LIN {X 0,Y 671.666,Z 913.822,A -85,B 0,C 180,E1 31372.923,E2 31372.923} C_VEL
LIN {X 0,Y 672.94,Z 893.638,A -85,B 0,C 180,E1 31372.091,E2 31372.091} C_VEL
LIN {X 0,Y 674.079,Z 873.149,A -85,B 0,C 180,E1 31371.357,E2 31371.357} C_VEL
LIN {X 0,Y 675.288,Z 850.138,A -85,B 0,C 180,E1 31370.661,E2 31370.661} C_VEL
LIN {X 0,Y 676.492,Z 822.718,A -85,B 0,C 180,E1 31370.003,E2 31370.003} C_VEL
LIN {X 0,Y 677.288,Z 796.769,A -85,B 0,C 180,E1 31369.548,E2 31369.548} C_VEL
LIN {X 0,Y 680.414,Z 579.65,A -85,B 0,C 180,E1 31366.739,E2 31366.739} C_VEL
LIN {X 0,Y 683.518,Z 369.829,A -85,B 0,C 180,E1 31363.955,E2 31363.955} C_VEL
LIN {X 0,Y 683.506,Z 361.175,A -85,B 0,C 180,E1 31363.826,E2 31363.826} C_VEL
LIN {X 0,Y 671.201,Z 343.19,A -85,B 0,C 180,E1 31362.442,E2 31362.442} C_VEL
LIN {X 0,Y 666.717,Z 337.316,A -85,B 0,C 180,E1 31361.923,E2 31361.923} C_VEL
LIN {X 0,Y 663.783,Z 333.148,A -85,B 0,C 180,E1 31361.571,E2 31361.571} C_VEL
LIN {X 0,Y 661.006,Z 329.319,A -85,B 0,C 180,E1 31361.235,E2 31361.235} C_VEL
LIN {X 0,Y 660.134,Z 328.105,A -85,B 0,C 180,E1 31361.129,E2 31361.129} C_VEL
LIN {X 0,Y 657.606,Z 325.421,A -85,B 0,C 180,E1 31360.83,E2 31360.83} C_VEL
LIN {X 0,Y 656.61,Z 322.443,A -85,B 0,C 180,E1 31360.675,E2 31360.675} C_VEL
LIN {X 0,Y 656.617,Z 322.441,A -85,B 0,C 180,E1 31358.189,E2 31358.189} C_VEL
LIN {X 0,Y 656.632,Z 322.413,A -85,B 0,C 180,E1 31355.035,E2 31355.035} C_VEL
LIN {X 0,Y 656.601,Z 322.44,A -85,B 0,C 180,E1 31352.311,E2 31352.311} C_VEL
LIN {X 0,Y 656.685,Z 322.411,A -85,B 0,C 180,E1 31349.435,E2 31349.435} C_VEL
LIN {X 0,Y 656.609,Z 322.425,A -85,B 0,C 180,E1 31346.443,E2 31346.443} C_VEL
LIN {X 0,Y 656.627,Z 322.43,A -85,B 0,C 180,E1 31343.799,E2 31343.799} C_VEL
LIN {X 0,Y 656.633,Z 322.407,A -85,B 0,C 180,E1 31340.595,E2 31340.595} C_VEL
LIN {X 0,Y 656.618,Z 322.434,A -85,B 0,C 180,E1 31338.007,E2 31338.007} C_VEL
LIN {X 0,Y 656.701,Z 322.403,A -85,B 0,C 180,E1 31335.092,E2 31335.092} C_VEL
LIN {X 0,Y 656.627,Z 322.434,A -85,B 0,C 180,E1 31332.131,E2 31332.131} C_VEL
LIN {X 0,Y 656.642,Z 322.414,A -85,B 0,C 180,E1 31329.466,E2 31329.466} C_VEL
LIN {X 0,Y 656.646,Z 322.432,A -85,B 0,C 180,E1 31326.207,E2 31326.207} C_VEL
LIN {X 0,Y 656.634,Z 322.418,A -85,B 0,C 180,E1 31323.579,E2 31323.579} C_VEL
LIN {X 0,Y 656.71,Z 322.429,A -85,B 0,C 180,E1 31320.523,E2 31320.523} C_VEL
LIN {X 0,Y 656.638,Z 322.42,A -85,B 0,C 180,E1 31317.644,E2 31317.644} C_VEL
LIN {X 0,Y 656.706,Z 322.421,A -85,B 0,C 180,E1 31314.706,E2 31314.706} C_VEL
LIN {X 0,Y 656.648,Z 322.417,A -85,B 0,C 180,E1 31311.682,E2 31311.682} C_VEL
LIN {X 0,Y 656.68,Z 322.422,A -85,B 0,C 180,E1 31308.85,E2 31308.85} C_VEL
LIN {X 0,Y 656.663,Z 322.41,A -85,B 0,C 180,E1 31305.719,E2 31305.719} C_VEL
LIN {X 0,Y 656.668,Z 322.428,A -85,B 0,C 180,E1 31302.91,E2 31302.91} C_VEL
LIN {X 0,Y 656.678,Z 322.403,A -85,B 0,C 180,E1 31299.686,E2 31299.686} C_VEL
LIN {X 0,Y 656.674,Z 322.435,A -85,B 0,C 180,E1 31296.773,E2 31296.773} C_VEL
LIN {X 0,Y 656.686,Z 322.424,A -85,B 0,C 180,E1 31293.544,E2 31293.544} C_VEL
LIN {X 0,Y 656.685,Z 322.409,A -85,B 0,C 180,E1 31290.54,E2 31290.54} C_VEL
LIN {X 0,Y 656.686,Z 322.425,A -85,B 0,C 180,E1 31287.35,E2 31287.35} C_VEL
LIN {X 0,Y 656.698,Z 322.433,A -85,B 0,C 180,E1 31284.327,E2 31284.327} C_VEL
LIN {X 0,Y 656.736,Z 322.619,A -85,B 0,C 180,E1 31281.555,E2 31281.555} C_VEL
LIN {X 0,Y 658.039,Z 325.986,A -85,B 0,C 180,E1 31281.13,E2 31281.13} C_VEL
LIN {X 0,Y 659.196,Z 328.329,A -85,B 0,C 180,E1 31280.812,E2 31280.812} C_VEL
LIN {X 0,Y 663.314,Z 336.664,A -85,B 0,C 180,E1 31279.705,E2 31279.705} C_VEL
LIN {X 0,Y 670.239,Z 350.9,A -85,B 0,C 180,E1 31277.945,E2 31277.945} C_VEL
LIN {X 0,Y 680.871,Z 366.63,A -85,B 0,C 180,E1 31276.729,E2 31276.729} C_VEL
LIN {X 0,Y 683.852,Z 379.489,A -85,B 0,C 180,E1 31276.273,E2 31276.273} C_VEL
LIN {X 0,Y 680.729,Z 587.028,A -85,B 0,C 180,E1 31273.513,E2 31273.513} C_VEL
LIN {X 0,Y 677.649,Z 809.677,A -85,B 0,C 180,E1 31270.64,E2 31270.64} C_VEL
LIN {X 0,Y 676.889,Z 840.625,A -85,B 0,C 180,E1 31270.183,E2 31270.183} C_VEL
LIN {X 0,Y 675.965,Z 864.916,A -85,B 0,C 180,E1 31269.679,E2 31269.679} C_VEL
LIN {X 0,Y 674.842,Z 889.591,A -85,B 0,C 180,E1 31269.027,E2 31269.027} C_VEL
LIN {X 0,Y 673.329,Z 917.024,A -85,B 0,C 180,E1 31268.116,E2 31268.116} C_VEL
LIN {X 0,Y 671.946,Z 939.064,A -85,B 0,C 180,E1 31267.24,E2 31267.24} C_VEL
LIN {X 0,Y 670.562,Z 959.722,A -85,B 0,C 180,E1 31266.296,E2 31266.296} C_VEL
LIN {X 0,Y 669.028,Z 981.503,A -85,B 0,C 180,E1 31265.163,E2 31265.163} C_VEL
LIN {X 0,Y 667.169,Z 1006.405,A -85,B 0,C 180,E1 31263.676,E2 31263.676} C_VEL
LIN {X 0,Y 665.527,Z 1027.238,A -85,B 0,C 180,E1 31262.257,E2 31262.257} C_VEL
LIN {X 0,Y 664.066,Z 1046.482,A -85,B 0,C 180,E1 31260.792,E2 31260.792} C_VEL
LIN {X 0,Y 662.377,Z 1069.251,A -85,B 0,C 180,E1 31258.835,E2 31258.835} C_VEL
LIN {X 0,Y 661.095,Z 1086.391,A -85,B 0,C 180,E1 31257.178,E2 31257.178} C_VEL
LIN {X 0,Y 659.976,Z 1103.08,A -85,B 0,C 180,E1 31255.388,E2 31255.388} C_VEL
LIN {X 0,Y 658.84,Z 1120.853,A -85,B 0,C 180,E1 31253.24,E2 31253.24} C_VEL
LIN {X 0,Y 658.05,Z 1134.796,A -85,B 0,C 180,E1 31251.339,E2 31251.339} C_VEL
LIN {X 0,Y 657.408,Z 1147.739,A -85,B 0,C 180,E1 31249.363,E2 31249.363} C_VEL
LIN {X 0,Y 656.816,Z 1161.282,A -85,B 0,C 180,E1 31246.994,E2 31246.994} C_VEL
LIN {X 0,Y 656.46,Z 1171.486,A -85,B 0,C 180,E1 31244.916,E2 31244.916} C_VEL
LIN {X 0,Y 656.243,Z 1179.514,A -85,B 0,C 180,E1 31243.032,E2 31243.032} C_VEL
LIN {X 0,Y 656.056,Z 1187.306,A -85,B 0,C 180,E1 31240.893,E2 31240.893} C_VEL
LIN {X 0,Y 655.979,Z 1194.036,A -85,B 0,C 180,E1 31238.591,E2 31238.591} C_VEL
LIN {X 0,Y 655.933,Z 1199.09,A -85,B 0,C 180,E1 31236.301,E2 31236.301} C_VEL
LIN {X 0,Y 655.917,Z 1202.479,A -85,B 0,C 180,E1 31234.108,E2 31234.108} C_VEL
LIN {X 0,Y 655.907,Z 1204.549,A -85,B 0,C 180,E1 31231.747,E2 31231.747} C_VEL
LIN {X 0,Y 655.891,Z 1204.872,A -85,B 0,C 180,E1 31229.476,E2 31229.476} C_VEL
LIN {X 0,Y 655.908,Z 1203.947,A -85,B 0,C 180,E1 31227.379,E2 31227.379} C_VEL
LIN {X 0,Y 655.919,Z 1201.428,A -85,B 0,C 180,E1 31225.103,E2 31225.103} C_VEL
LIN {X 0,Y 655.949,Z 1197.152,A -85,B 0,C 180,E1 31222.732,E2 31222.732} C_VEL
LIN {X 0,Y 656.009,Z 1191.376,A -85,B 0,C 180,E1 31220.437,E2 31220.437} C_VEL
LIN {X 0,Y 656.126,Z 1184.279,A -85,B 0,C 180,E1 31218.217,E2 31218.217} C_VEL
LIN {X 0,Y 656.39,Z 1174.089,A -85,B 0,C 180,E1 31215.658,E2 31215.658} C_VEL
LIN {X 0,Y 656.694,Z 1164.273,A -85,B 0,C 180,E1 31213.587,E2 31213.587} C_VEL
LIN {X 0,Y 657.112,Z 1154.137,A -85,B 0,C 180,E1 31211.716,E2 31211.716} C_VEL
LIN {X 0,Y 657.764,Z 1140.78,A -85,B 0,C 180,E1 31209.536,E2 31209.536} C_VEL
LIN {X 0,Y 658.6,Z 1125.104,A -85,B 0,C 180,E1 31207.318,E2 31207.318} C_VEL
LIN {X 0,Y 659.476,Z 1110.399,A -85,B 0,C 180,E1 31205.467,E2 31205.467} C_VEL
LIN {X 0,Y 660.73,Z 1092.314,A -85,B 0,C 180,E1 31203.428,E2 31203.428} C_VEL
LIN {X 0,Y 662,Z 1073.819,A -85,B 0,C 180,E1 31201.591,E2 31201.591} C_VEL
LIN {X 0,Y 663.289,Z 1056.842,A -85,B 0,C 180,E1 31200.069,E2 31200.069} C_VEL
LIN {X 0,Y 664.963,Z 1035.53,A -85,B 0,C 180,E1 31198.348,E2 31198.348} C_VEL
LIN {X 0,Y 666.618,Z 1013.004,A -85,B 0,C 180,E1 31196.756,E2 31196.756} C_VEL
LIN {X 0,Y 668.131,Z 993.022,A -85,B 0,C 180,E1 31195.499,E2 31195.499} C_VEL
LIN {X 0,Y 669.972,Z 968.967,A -85,B 0,C 180,E1 31194.161,E2 31194.161} C_VEL
LIN {X 0,Y 671.656,Z 944.002,A -85,B 0,C 180,E1 31192.976,E2 31192.976} C_VEL
LIN {X 0,Y 672.974,Z 923.056,A -85,B 0,C 180,E1 31192.114,E2 31192.114} C_VEL
LIN {X 0,Y 674.098,Z 902.837,A -85,B 0,C 180,E1 31191.392,E2 31191.392} C_VEL
LIN {X 0,Y 675.317,Z 879.538,A -85,B 0,C 180,E1 31190.689,E2 31190.689} C_VEL
LIN {X 0,Y 676.525,Z 851.65,A -85,B 0,C 180,E1 31190.026,E2 31190.026} C_VEL
LIN {X 0,Y 677.299,Z 826.243,A -85,B 0,C 180,E1 31189.585,E2 31189.585} C_VEL
LIN {X 0,Y 680.398,Z 610.207,A -85,B 0,C 180,E1 31186.79,E2 31186.79} C_VEL
LIN {X 0,Y 683.523,Z 400.862,A -85,B 0,C 180,E1 31184.016,E2 31184.016} C_VEL
LIN {X 0,Y 683.703,Z 378.044,A -85,B 0,C 180,E1 31183.693,E2 31183.693} C_VEL
LIN {X 0,Y 680.509,Z 365.883,A -85,B 0,C 180,E1 31183.227,E2 31183.227} C_VEL
LIN {X 0,Y 669.705,Z 349.983,A -85,B 0,C 180,E1 31181.969,E2 31181.969} C_VEL
LIN {X 0,Y 661.964,Z 333.955,A -85,B 0,C 180,E1 31179.938,E2 31179.938} C_VEL
LIN {X 0,Y 659.979,Z 329.954,A -85,B 0,C 180,E1 31179.405,E2 31179.405} C_VEL
LIN {X 0,Y 658.426,Z 326.508,A -85,B 0,C 180,E1 31178.955,E2 31178.955} C_VEL
LIN {X 0,Y 656.846,Z 323.199,A -85,B 0,C 180,E1 31178.507,E2 31178.507} C_VEL
LIN {X 0,Y 656.707,Z 322.413,A -85,B 0,C 180,E1 31178.405,E2 31178.405} C_VEL
LIN {X 0,Y 656.675,Z 322.429,A -85,B 0,C 180,E1 31175.302,E2 31175.302} C_VEL
LIN {X 0,Y 656.707,Z 322.423,A -85,B 0,C 180,E1 31172.305,E2 31172.305} C_VEL
LIN {X 0,Y 656.672,Z 322.412,A -85,B 0,C 180,E1 31169.255,E2 31169.255} C_VEL
LIN {X 0,Y 656.703,Z 322.418,A -85,B 0,C 180,E1 31166.263,E2 31166.263} C_VEL
LIN {X 0,Y 656.672,Z 322.434,A -85,B 0,C 180,E1 31163.124,E2 31163.124} C_VEL
LIN {X 0,Y 656.698,Z 322.401,A -85,B 0,C 180,E1 31160.127,E2 31160.127} C_VEL
LIN {X 0,Y 656.666,Z 322.429,A -85,B 0,C 180,E1 31156.999,E2 31156.999} C_VEL
LIN {X 0,Y 656.682,Z 322.407,A -85,B 0,C 180,E1 31154.096,E2 31154.096} C_VEL
LIN {X 0,Y 656.668,Z 322.424,A -85,B 0,C 180,E1 31150.972,E2 31150.972} C_VEL
LIN {X 0,Y 656.659,Z 322.414,A -85,B 0,C 180,E1 31148.141,E2 31148.141} C_VEL
LIN {X 0,Y 656.677,Z 322.422,A -85,B 0,C 180,E1 31144.979,E2 31144.979} C_VEL
LIN {X 0,Y 656.646,Z 322.416,A -85,B 0,C 180,E1 31142.182,E2 31142.182} C_VEL
LIN {X 0,Y 656.705,Z 322.424,A -85,B 0,C 180,E1 31139.128,E2 31139.128} C_VEL
LIN {X 0,Y 656.635,Z 322.417,A -85,B 0,C 180,E1 31136.246,E2 31136.246} C_VEL
LIN {X 0,Y 656.699,Z 322.43,A -85,B 0,C 180,E1 31133.355,E2 31133.355} C_VEL
LIN {X 0,Y 656.637,Z 322.414,A -85,B 0,C 180,E1 31130.357,E2 31130.357} C_VEL
LIN {X 0,Y 656.64,Z 322.433,A -85,B 0,C 180,E1 31127.691,E2 31127.691} C_VEL
LIN {X 0,Y 656.66,Z 322.411,A -85,B 0,C 180,E1 31124.543,E2 31124.543} C_VEL
LIN {X 0,Y 656.624,Z 322.434,A -85,B 0,C 180,E1 31121.81,E2 31121.81} C_VEL
LIN {X 0,Y 656.707,Z 322.404,A -85,B 0,C 180,E1 31118.847,E2 31118.847} C_VEL
LIN {X 0,Y 656.619,Z 322.43,A -85,B 0,C 180,E1 31115.914,E2 31115.914} C_VEL
LIN {X 0,Y 656.63,Z 322.422,A -85,B 0,C 180,E1 31113.307,E2 31113.307} C_VEL
LIN {X 0,Y 656.637,Z 322.411,A -85,B 0,C 180,E1 31110.136,E2 31110.136} C_VEL
LIN {X 0,Y 656.609,Z 322.439,A -85,B 0,C 180,E1 31107.523,E2 31107.523} C_VEL
LIN {X 0,Y 656.676,Z 322.411,A -85,B 0,C 180,E1 31104.647,E2 31104.647} C_VEL
LIN {X 0,Y 656.604,Z 322.415,A -85,B 0,C 180,E1 31101.649,E2 31101.649} C_VEL
LIN {X 0,Y 656.688,Z 322.418,A -85,B 0,C 180,E1 31100.473,E2 31100.473} C_VEL
LIN {X 0,Y 656.825,Z 323.195,A -85,B 0,C 180,E1 31100.104,E2 31100.104} C_VEL
LIN {X 0,Y 657.18,Z 325.756,A -85,B 0,C 180,E1 31099.685,E2 31099.685} C_VEL
LIN {X 0,Y 658.094,Z 331.001,A -85,B 0,C 180,E1 31099.187,E2 31099.187} C_VEL
LIN {X 0,Y 660.809,Z 339.923,A -85,B 0,C 180,E1 31098.553,E2 31098.553} C_VEL
LIN {X 0,Y 663.684,Z 344.552,A -85,B 0,C 180,E1 31098.166,E2 31098.166} C_VEL
LIN {X 0,Y 670.686,Z 354.26,A -85,B 0,C 180,E1 31097.344,E2 31097.344} C_VEL
LIN {X 0,Y 678.016,Z 365.563,A -85,B 0,C 180,E1 31096.503,E2 31096.503} C_VEL
LIN {X 0,Y 674.796,Z 565.744,A -85,B 0,C 180,E1 31093.822,E2 31093.822} C_VEL
LIN {X 0,Y 671.317,Z 791.977,A -85,B 0,C 180,E1 31090.876,E2 31090.876} C_VEL
LIN {X 0,Y 670.56,Z 815.572,A -85,B 0,C 180,E1 31090.489,E2 31090.489} C_VEL
LIN {X 0,Y 669.499,Z 841.04,A -85,B 0,C 180,E1 31089.93,E2 31089.93} C_VEL
LIN {X 0,Y 668.036,Z 868.498,A -85,B 0,C 180,E1 31089.141,E2 31089.141} C_VEL
LIN {X 0,Y 666.707,Z 890.267,A -85,B 0,C 180,E1 31088.38,E2 31088.38} C_VEL
LIN {X 0,Y 665.306,Z 910.812,A -85,B 0,C 180,E1 31087.547,E2 31087.547} C_VEL
LIN {X 0,Y 663.778,Z 931.891,A -85,B 0,C 180,E1 31086.566,E2 31086.566} C_VEL
LIN {X 0,Y 661.891,Z 956.652,A -85,B 0,C 180,E1 31085.243,E2 31085.243} C_VEL
LIN {X 0,Y 659.976,Z 979.437,A -85,B 0,C 180,E1 31083.832,E2 31083.832} C_VEL
LIN {X 0,Y 658.322,Z 998.997,A -85,B 0,C 180,E1 31082.472,E2 31082.472} C_VEL
LIN {X 0,Y 656.56,Z 1020.781,A -85,B 0,C 180,E1 31080.776,E2 31080.776} C_VEL
LIN {X 0,Y 654.855,Z 1041.333,A -85,B 0,C 180,E1 31078.947,E2 31078.947} C_VEL
LIN {X 0,Y 653.526,Z 1057.819,A -85,B 0,C 180,E1 31077.321,E2 31077.321} C_VEL
LIN {X 0,Y 652.214,Z 1076.039,A -85,B 0,C 180,E1 31075.322,E2 31075.322} C_VEL
LIN {X 0,Y 651.029,Z 1092.653,A -85,B 0,C 180,E1 31073.247,E2 31073.247} C_VEL
LIN {X 0,Y 650.204,Z 1106.086,A -85,B 0,C 180,E1 31071.374,E2 31071.374} C_VEL
LIN {X 0,Y 649.455,Z 1120.323,A -85,B 0,C 180,E1 31069.143,E2 31069.143} C_VEL
LIN {X 0,Y 648.84,Z 1132.921,A -85,B 0,C 180,E1 31066.84,E2 31066.84} C_VEL
LIN {X 0,Y 648.504,Z 1142.107,A -85,B 0,C 180,E1 31064.92,E2 31064.92} C_VEL
LIN {X 0,Y 648.255,Z 1150.555,A -85,B 0,C 180,E1 31062.884,E2 31062.884} C_VEL
LIN {X 0,Y 648.065,Z 1158.619,A -85,B 0,C 180,E1 31060.579,E2 31060.579} C_VEL
LIN {X 0,Y 647.974,Z 1165.226,A -85,B 0,C 180,E1 31058.161,E2 31058.161} C_VEL
LIN {X 0,Y 647.931,Z 1169.805,A -85,B 0,C 180,E1 31055.934,E2 31055.934} C_VEL
LIN {X 0,Y 647.913,Z 1173.144,A -85,B 0,C 180,E1 31053.539,E2 31053.539} C_VEL
LIN {X 0,Y 647.91,Z 1174.68,A -85,B 0,C 180,E1 31051.238,E2 31051.238} C_VEL
LIN {X 0,Y 647.896,Z 1174.838,A -85,B 0,C 180,E1 31049.293,E2 31049.293} C_VEL
LIN {X 0,Y 647.909,Z 1173.911,A -85,B 0,C 180,E1 31047.258,E2 31047.258} C_VEL
LIN {X 0,Y 647.921,Z 1171.367,A -85,B 0,C 180,E1 31044.954,E2 31044.954} C_VEL
LIN {X 0,Y 647.946,Z 1167.055,A -85,B 0,C 180,E1 31042.552,E2 31042.552} C_VEL
LIN {X 0,Y 648.019,Z 1161.246,A -85,B 0,C 180,E1 31040.228,E2 31040.228} C_VEL
LIN {X 0,Y 648.159,Z 1153.801,A -85,B 0,C 180,E1 31037.89,E2 31037.89} C_VEL
LIN {X 0,Y 648.461,Z 1143.728,A -85,B 0,C 180,E1 31035.353,E2 31035.353} C_VEL
LIN {X 0,Y 648.781,Z 1134.303,A -85,B 0,C 180,E1 31033.343,E2 31033.343} C_VEL
LIN {X 0,Y 649.238,Z 1123.964,A -85,B 0,C 180,E1 31031.41,E2 31031.41} C_VEL
LIN {X 0,Y 649.968,Z 1110.475,A -85,B 0,C 180,E1 31029.185,E2 31029.185} C_VEL
LIN {X 0,Y 650.893,Z 1094.731,A -85,B 0,C 180,E1 31026.939,E2 31026.939} C_VEL
LIN {X 0,Y 651.841,Z 1080.663,A -85,B 0,C 180,E1 31025.147,E2 31025.147} C_VEL
LIN {X 0,Y 653.205,Z 1062.368,A -85,B 0,C 180,E1 31023.058,E2 31023.058} C_VEL
LIN {X 0,Y 654.644,Z 1043.712,A -85,B 0,C 180,E1 31021.187,E2 31021.187} C_VEL
LIN {X 0,Y 656.036,Z 1026.779,A -85,B 0,C 180,E1 31019.653,E2 31019.653} C_VEL
LIN {X 0,Y 657.802,Z 1006.081,A -85,B 0,C 180,E1 31017.962,E2 31017.962} C_VEL
LIN {X 0,Y 659.644,Z 983.162,A -85,B 0,C 180,E1 31016.323,E2 31016.323} C_VEL
LIN {X 0,Y 661.323,Z 962.904,A -85,B 0,C 180,E1 31015.04,E2 31015.04} C_VEL
LIN {X 0,Y 663.335,Z 938.507,A -85,B 0,C 180,E1 31013.674,E2 31013.674} C_VEL
LIN {X 0,Y 665.121,Z 913.811,A -85,B 0,C 180,E1 31012.496,E2 31012.496} C_VEL
LIN {X 0,Y 666.501,Z 893.662,A -85,B 0,C 180,E1 31011.661,E2 31011.661} C_VEL
LIN {X 0,Y 667.739,Z 873.127,A -85,B 0,C 180,E1 31010.921,E2 31010.921} C_VEL
LIN {X 0,Y 669.012,Z 850.563,A -85,B 0,C 180,E1 31010.234,E2 31010.234} C_VEL
LIN {X 0,Y 670.3,Z 823.602,A -85,B 0,C 180,E1 31009.579,E2 31009.579} C_VEL
LIN {X 0,Y 671.173,Z 797.336,A -85,B 0,C 180,E1 31009.112,E2 31009.112} C_VEL
LIN {X 0,Y 674.494,Z 585.107,A -85,B 0,C 180,E1 31006.343,E2 31006.343} C_VEL
LIN {X 0,Y 677.899,Z 373.5,A -85,B 0,C 180,E1 31003.516,E2 31003.516} C_VEL
LIN {X 0,Y 677.911,Z 365.067,A -85,B 0,C 180,E1 31003.39,E2 31003.39} C_VEL
LIN {X 0,Y 667.133,Z 349.224,A -85,B 0,C 180,E1 31002.151,E2 31002.151} C_VEL
LIN {X 0,Y 659.308,Z 338.748,A -85,B 0,C 180,E1 31001.219,E2 31001.219} C_VEL
LIN {X 0,Y 656.27,Z 334.548,A -85,B 0,C 180,E1 31000.844,E2 31000.844} C_VEL
LIN {X 0,Y 653.322,Z 330.877,A -85,B 0,C 180,E1 31000.481,E2 31000.481} C_VEL
LIN {X 0,Y 652.237,Z 329.139,A -85,B 0,C 180,E1 31000.34,E2 31000.34} C_VEL
LIN {X 0,Y 649.752,Z 326.511,A -85,B 0,C 180,E1 31000.035,E2 31000.035} C_VEL
LIN {X 0,Y 648.72,Z 323.425,A -85,B 0,C 180,E1 30999.865,E2 30999.865} C_VEL
LIN {X 0,Y 648.678,Z 323.43,A -85,B 0,C 180,E1 30996.843,E2 30996.843} C_VEL
LIN {X 0,Y 648.663,Z 323.402,A -85,B 0,C 180,E1 30994.238,E2 30994.238} C_VEL
LIN {X 0,Y 648.729,Z 323.402,A -85,B 0,C 180,E1 30991.197,E2 30991.197} C_VEL
LIN {X 0,Y 648.669,Z 323.426,A -85,B 0,C 180,E1 30988.445,E2 30988.445} C_VEL
LIN {X 0,Y 648.686,Z 323.402,A -85,B 0,C 180,E1 30985.822,E2 30985.822} C_VEL
LIN {X 0,Y 648.69,Z 323.423,A -85,B 0,C 180,E1 30982.57,E2 30982.57} C_VEL
LIN {X 0,Y 648.675,Z 323.396,A -85,B 0,C 180,E1 30980.011,E2 30980.011} C_VEL
LIN {X 0,Y 648.766,Z 323.415,A -85,B 0,C 180,E1 30977.028,E2 30977.028} C_VEL
LIN {X 0,Y 648.682,Z 323.403,A -85,B 0,C 180,E1 30974.096,E2 30974.096} C_VEL
LIN {X 0,Y 648.717,Z 323.425,A -85,B 0,C 180,E1 30971.379,E2 30971.379} C_VEL
LIN {X 0,Y 648.702,Z 323.4,A -85,B 0,C 180,E1 30968.242,E2 30968.242} C_VEL
LIN {X 0,Y 648.697,Z 323.424,A -85,B 0,C 180,E1 30965.573,E2 30965.573} C_VEL
LIN {X 0,Y 648.748,Z 323.39,A -85,B 0,C 180,E1 30962.473,E2 30962.473} C_VEL
LIN {X 0,Y 648.698,Z 323.422,A -85,B 0,C 180,E1 30959.647,E2 30959.647} C_VEL
LIN {X 0,Y 648.763,Z 323.388,A -85,B 0,C 180,E1 30956.731,E2 30956.731} C_VEL
LIN {X 0,Y 648.708,Z 323.42,A -85,B 0,C 180,E1 30953.717,E2 30953.717} C_VEL
LIN {X 0,Y 648.74,Z 323.392,A -85,B 0,C 180,E1 30950.865,E2 30950.865} C_VEL
LIN {X 0,Y 648.722,Z 323.418,A -85,B 0,C 180,E1 30947.719,E2 30947.719} C_VEL
LIN {X 0,Y 648.728,Z 323.393,A -85,B 0,C 180,E1 30944.901,E2 30944.901} C_VEL
LIN {X 0,Y 648.734,Z 323.415,A -85,B 0,C 180,E1 30941.674,E2 30941.674} C_VEL
LIN {X 0,Y 648.736,Z 323.399,A -85,B 0,C 180,E1 30938.764,E2 30938.764} C_VEL
LIN {X 0,Y 648.744,Z 323.402,A -85,B 0,C 180,E1 30935.603,E2 30935.603} C_VEL
LIN {X 0,Y 648.751,Z 323.421,A -85,B 0,C 180,E1 30932.559,E2 30932.559} C_VEL
LIN {X 0,Y 648.738,Z 323.405,A -85,B 0,C 180,E1 30929.317,E2 30929.317} C_VEL
LIN {X 0,Y 648.759,Z 323.394,A -85,B 0,C 180,E1 30926.3,E2 30926.3} C_VEL
LIN {X 0,Y 648.739,Z 323.4,A -85,B 0,C 180,E1 30923.12,E2 30923.12} C_VEL
LIN {X 0,Y 648.774,Z 323.536,A -85,B 0,C 180,E1 30922.332,E2 30922.332} C_VEL
LIN {X 0,Y 649.998,Z 326.772,A -85,B 0,C 180,E1 30921.913,E2 30921.913} C_VEL
LIN {X 0,Y 651.055,Z 328.483,A -85,B 0,C 180,E1 30921.65,E2 30921.65} C_VEL
LIN {X 0,Y 659.144,Z 345.329,A -85,B 0,C 180,E1 30919.4,E2 30919.4} C_VEL
LIN {X 0,Y 661.685,Z 350.479,A -85,B 0,C 180,E1 30918.773,E2 30918.773} C_VEL
LIN {X 0,Y 675.933,Z 371.231,A -85,B 0,C 180,E1 30917.105,E2 30917.105} C_VEL
LIN {X 0,Y 678.28,Z 381.651,A -85,B 0,C 180,E1 30916.734,E2 30916.734} C_VEL
LIN {X 0,Y 674.888,Z 589.308,A -85,B 0,C 180,E1 30913.953,E2 30913.953} C_VEL
LIN {X 0,Y 671.538,Z 812.221,A -85,B 0,C 180,E1 30911.054,E2 30911.054} C_VEL
LIN {X 0,Y 670.725,Z 841.411,A -85,B 0,C 180,E1 30910.611,E2 30910.611} C_VEL
LIN {X 0,Y 669.756,Z 865.157,A -85,B 0,C 180,E1 30910.114,E2 30910.114} C_VEL
LIN {X 0,Y 668.563,Z 889.44,A -85,B 0,C 180,E1 30909.469,E2 30909.469} C_VEL
LIN {X 0,Y 666.876,Z 917.596,A -85,B 0,C 180,E1 30908.527,E2 30908.527} C_VEL
LIN {X 0,Y 665.363,Z 939.922,A -85,B 0,C 180,E1 30907.63,E2 30907.63} C_VEL
LIN {X 0,Y 663.854,Z 960.724,A -85,B 0,C 180,E1 30906.668,E2 30906.668} C_VEL
LIN {X 0,Y 662.096,Z 983.91,A -85,B 0,C 180,E1 30905.443,E2 30905.443} C_VEL
LIN {X 0,Y 660.055,Z 1008.607,A -85,B 0,C 180,E1 30903.932,E2 30903.932} C_VEL
LIN {X 0,Y 658.45,Z 1027.583,A -85,B 0,C 180,E1 30902.62,E2 30902.62} C_VEL
LIN {X 0,Y 656.822,Z 1047.088,A -85,B 0,C 180,E1 30901.118,E2 30901.118} C_VEL
LIN {X 0,Y 654.983,Z 1069.759,A -85,B 0,C 180,E1 30899.141,E2 30899.141} C_VEL
LIN {X 0,Y 653.646,Z 1086.39,A -85,B 0,C 180,E1 30897.513,E2 30897.513} C_VEL
LIN {X 0,Y 652.369,Z 1103.306,A -85,B 0,C 180,E1 30895.679,E2 30895.679} C_VEL
LIN {X 0,Y 651.106,Z 1121.566,A -85,B 0,C 180,E1 30893.436,E2 30893.436} C_VEL
LIN {X 0,Y 650.245,Z 1135.429,A -85,B 0,C 180,E1 30891.515,E2 30891.515} C_VEL
LIN {X 0,Y 649.487,Z 1149.548,A -85,B 0,C 180,E1 30889.313,E2 30889.313} C_VEL
LIN {X 0,Y 648.875,Z 1162.214,A -85,B 0,C 180,E1 30887.024,E2 30887.024} C_VEL
LIN {X 0,Y 648.512,Z 1171.487,A -85,B 0,C 180,E1 30885.103,E2 30885.103} C_VEL
LIN {X 0,Y 648.28,Z 1179.515,A -85,B 0,C 180,E1 30883.195,E2 30883.195} C_VEL
LIN {X 0,Y 648.084,Z 1187.034,A -85,B 0,C 180,E1 30881.112,E2 30881.112} C_VEL
LIN {X 0,Y 647.987,Z 1193.816,A -85,B 0,C 180,E1 30878.787,E2 30878.787} C_VEL
LIN {X 0,Y 647.935,Z 1199.101,A -85,B 0,C 180,E1 30876.372,E2 30876.372} C_VEL
LIN {X 0,Y 647.918,Z 1202.476,A -85,B 0,C 180,E1 30874.159,E2 30874.159} C_VEL
LIN {X 0,Y 647.907,Z 1204.549,A -85,B 0,C 180,E1 30871.769,E2 30871.769} C_VEL
LIN {X 0,Y 647.892,Z 1204.872,A -85,B 0,C 180,E1 30869.469,E2 30869.469} C_VEL
LIN {X 0,Y 647.909,Z 1203.944,A -85,B 0,C 180,E1 30867.346,E2 30867.346} C_VEL
LIN {X 0,Y 647.922,Z 1201.427,A -85,B 0,C 180,E1 30865.042,E2 30865.042} C_VEL
LIN {X 0,Y 647.951,Z 1197.151,A -85,B 0,C 180,E1 30862.641,E2 30862.641} C_VEL
LIN {X 0,Y 648.018,Z 1191.373,A -85,B 0,C 180,E1 30860.318,E2 30860.318} C_VEL
LIN {X 0,Y 648.146,Z 1184.279,A -85,B 0,C 180,E1 30858.07,E2 30858.07} C_VEL
LIN {X 0,Y 648.439,Z 1174.338,A -85,B 0,C 180,E1 30855.535,E2 30855.535} C_VEL
LIN {X 0,Y 648.771,Z 1164.544,A -85,B 0,C 180,E1 30853.434,E2 30853.434} C_VEL
LIN {X 0,Y 649.238,Z 1154.237,A -85,B 0,C 180,E1 30851.503,E2 30851.503} C_VEL
LIN {X 0,Y 649.924,Z 1141.364,A -85,B 0,C 180,E1 30849.372,E2 30849.372} C_VEL
LIN {X 0,Y 650.838,Z 1125.803,A -85,B 0,C 180,E1 30847.128,E2 30847.128} C_VEL
LIN {X 0,Y 651.804,Z 1111.152,A -85,B 0,C 180,E1 30845.252,E2 30845.252} C_VEL
LIN {X 0,Y 653.113,Z 1093.727,A -85,B 0,C 180,E1 30843.251,E2 30843.251} C_VEL
LIN {X 0,Y 654.547,Z 1074.832,A -85,B 0,C 180,E1 30841.337,E2 30841.337} C_VEL
LIN {X 0,Y 655.937,Z 1057.951,A -85,B 0,C 180,E1 30839.8,E2 30839.8} C_VEL
LIN {X 0,Y 657.511,Z 1039.194,A -85,B 0,C 180,E1 30838.254,E2 30838.254} C_VEL
LIN {X 0,Y 659.486,Z 1015.133,A -85,B 0,C 180,E1 30836.501,E2 30836.501} C_VEL
LIN {X 0,Y 661.141,Z 994.951,A -85,B 0,C 180,E1 30835.207,E2 30835.207} C_VEL
LIN {X 0,Y 662.831,Z 974.061,A -85,B 0,C 180,E1 30834.017,E2 30834.017} C_VEL
LIN {X 0,Y 664.822,Z 948.476,A -85,B 0,C 180,E1 30832.747,E2 30832.747} C_VEL
LIN {X 0,Y 666.407,Z 925.175,A -85,B 0,C 180,E1 30831.764,E2 30831.764} C_VEL
LIN {X 0,Y 667.661,Z 904.466,A -85,B 0,C 180,E1 30831.01,E2 30831.01} C_VEL
LIN {X 0,Y 668.911,Z 882.309,A -85,B 0,C 180,E1 30830.328,E2 30830.328} C_VEL
LIN {X 0,Y 670.161,Z 856.684,A -85,B 0,C 180,E1 30829.689,E2 30829.689} C_VEL
LIN {X 0,Y 671.133,Z 829.116,A -85,B 0,C 180,E1 30829.183,E2 30829.183} C_VEL
LIN {X 0,Y 672.991,Z 713.103,A -85,B 0,C 180,E1 30827.667,E2 30827.667} C_VEL
LIN {X 0,Y 676.466,Z 491.125,A -85,B 0,C 180,E1 30824.743,E2 30824.743} C_VEL
LIN {X 0,Y 678.142,Z 380.284,A -85,B 0,C 180,E1 30823.233,E2 30823.233} C_VEL
LIN {X 0,Y 675.637,Z 370.746,A -85,B 0,C 180,E1 30822.86,E2 30822.86} C_VEL
LIN {X 0,Y 661.182,Z 349.497,A -85,B 0,C 180,E1 30821.136,E2 30821.136} C_VEL
LIN {X 0,Y 654.178,Z 335.204,A -85,B 0,C 180,E1 30819.256,E2 30819.256} C_VEL
LIN {X 0,Y 652.233,Z 331.232,A -85,B 0,C 180,E1 30818.714,E2 30818.714} C_VEL
LIN {X 0,Y 650.37,Z 327.299,A -85,B 0,C 180,E1 30818.174,E2 30818.174} C_VEL
LIN {X 0,Y 648.857,Z 323.994,A -85,B 0,C 180,E1 30817.718,E2 30817.718} C_VEL
LIN {X 0,Y 648.749,Z 323.394,A -85,B 0,C 180,E1 30817.61,E2 30817.61} C_VEL
LIN {X 0,Y 648.759,Z 323.399,A -85,B 0,C 180,E1 30814.554,E2 30814.554} C_VEL
LIN {X 0,Y 648.742,Z 323.416,A -85,B 0,C 180,E1 30811.369,E2 30811.369} C_VEL
LIN {X 0,Y 648.766,Z 323.408,A -85,B 0,C 180,E1 30808.34,E2 30808.34} C_VEL
LIN {X 0,Y 648.731,Z 323.395,A -85,B 0,C 180,E1 30805.176,E2 30805.176} C_VEL
LIN {X 0,Y 648.768,Z 323.416,A -85,B 0,C 180,E1 30802.145,E2 30802.145} C_VEL
LIN {X 0,Y 648.724,Z 323.41,A -85,B 0,C 180,E1 30798.979,E2 30798.979} C_VEL
LIN {X 0,Y 648.759,Z 323.405,A -85,B 0,C 180,E1 30796.015,E2 30796.015} C_VEL
LIN {X 0,Y 648.724,Z 323.422,A -85,B 0,C 180,E1 30792.914,E2 30792.914} C_VEL
LIN {X 0,Y 648.737,Z 323.403,A -85,B 0,C 180,E1 30790.03,E2 30790.03} C_VEL
LIN {X 0,Y 648.722,Z 323.423,A -85,B 0,C 180,E1 30786.816,E2 30786.816} C_VEL
LIN {X 0,Y 648.716,Z 323.405,A -85,B 0,C 180,E1 30784.066,E2 30784.066} C_VEL
LIN {X 0,Y 648.736,Z 323.421,A -85,B 0,C 180,E1 30780.883,E2 30780.883} C_VEL
LIN {X 0,Y 648.7,Z 323.407,A -85,B 0,C 180,E1 30778.145,E2 30778.145} C_VEL
LIN {X 0,Y 648.77,Z 323.407,A -85,B 0,C 180,E1 30775.137,E2 30775.137} C_VEL
LIN {X 0,Y 648.697,Z 323.408,A -85,B 0,C 180,E1 30772.204,E2 30772.204} C_VEL
LIN {X 0,Y 648.743,Z 323.406,A -85,B 0,C 180,E1 30769.342,E2 30769.342} C_VEL
LIN {X 0,Y 648.695,Z 323.407,A -85,B 0,C 180,E1 30766.268,E2 30766.268} C_VEL
LIN {X 0,Y 648.696,Z 323.413,A -85,B 0,C 180,E1 30763.616,E2 30763.616} C_VEL
LIN {X 0,Y 648.718,Z 323.4,A -85,B 0,C 180,E1 30760.46,E2 30760.46} C_VEL
LIN {X 0,Y 648.68,Z 323.422,A -85,B 0,C 180,E1 30757.812,E2 30757.812} C_VEL
LIN {X 0,Y 648.714,Z 323.405,A -85,B 0,C 180,E1 30755.116,E2 30755.116} C_VEL
LIN {X 0,Y 648.688,Z 323.427,A -85,B 0,C 180,E1 30752.03,E2 30752.03} C_VEL
LIN {X 0,Y 648.672,Z 323.399,A -85,B 0,C 180,E1 30749.501,E2 30749.501} C_VEL
LIN {X 0,Y 648.748,Z 323.409,A -85,B 0,C 180,E1 30746.617,E2 30746.617} C_VEL
LIN {X 0,Y 648.668,Z 323.43,A -85,B 0,C 180,E1 30743.597,E2 30743.597} C_VEL
LIN {X 0,Y 648.68,Z 323.404,A -85,B 0,C 180,E1 30740.973,E2 30740.973} C_VEL
LIN {X 0,Y 648.736,Z 323.658,A -85,B 0,C 180,E1 30740.031,E2 30740.031} C_VEL
LIN {X 0,Y 649.942,Z 326.839,A -85,B 0,C 180,E1 30739.849,E2 30739.849} C_VEL
LIN {X 0,Y 652.798,Z 329.833,A -85,B 0,C 180,E1 30739.5,E2 30739.5} C_VEL
LIN {X 0,Y 655.355,Z 333.679,A -85,B 0,C 180,E1 30739.173,E2 30739.173} C_VEL
LIN {X 0,Y 657.199,Z 335.747,A -85,B 0,C 180,E1 30738.952,E2 30738.952} C_VEL
LIN {X 0,Y 663.684,Z 344.552,A -85,B 0,C 180,E1 30738.166,E2 30738.166} C_VEL
LIN {X 0,Y 665.429,Z 347.736,A -85,B 0,C 180,E1 30737.946,E2 30737.946} C_VEL
LIN {X 0,Y 666.945,Z 354.539,A -85,B 0,C 180,E1 30737.693,E2 30737.693} C_VEL
LIN {X 0,Y 668.499,Z 362.251,A -85,B 0,C 180,E1 30737.425,E2 30737.425} C_VEL
LIN {X 0,Y 669.837,Z 365.18,A -85,B 0,C 180,E1 30737.254,E2 30737.254} C_VEL
LIN {X 0,Y 672.446,Z 369.387,A -85,B 0,C 180,E1 30736.947,E2 30736.947} C_VEL
LIN {X 0,Y 668.922,Z 571.887,A -85,B 0,C 180,E1 30734.217,E2 30734.217} C_VEL
LIN {X 0,Y 665.227,Z 793.273,A -85,B 0,C 180,E1 30731.31,E2 30731.31} C_VEL
LIN {X 0,Y 664.424,Z 816.456,A -85,B 0,C 180,E1 30730.923,E2 30730.923} C_VEL
LIN {X 0,Y 663.246,Z 842.682,A -85,B 0,C 180,E1 30730.338,E2 30730.338} C_VEL
LIN {X 0,Y 661.712,Z 869.106,A -85,B 0,C 180,E1 30729.566,E2 30729.566} C_VEL
LIN {X 0,Y 660.316,Z 890.28,A -85,B 0,C 180,E1 30728.82,E2 30728.82} C_VEL
LIN {X 0,Y 658.809,Z 910.823,A -85,B 0,C 180,E1 30727.982,E2 30727.982} C_VEL
LIN {X 0,Y 657.091,Z 932.902,A -85,B 0,C 180,E1 30726.945,E2 30726.945} C_VEL
LIN {X 0,Y 654.935,Z 958.727,A -85,B 0,C 180,E1 30725.537,E2 30725.537} C_VEL
LIN {X 0,Y 653.011,Z 980.178,A -85,B 0,C 180,E1 30724.189,E2 30724.189} C_VEL
LIN {X 0,Y 651.323,Z 998.723,A -85,B 0,C 180,E1 30722.887,E2 30722.887} C_VEL
LIN {X 0,Y 649.407,Z 1020.188,A -85,B 0,C 180,E1 30721.204,E2 30721.204} C_VEL
LIN {X 0,Y 647.564,Z 1040.832,A -85,B 0,C 180,E1 30719.356,E2 30719.356} C_VEL
LIN {X 0,Y 646.146,Z 1057.185,A -85,B 0,C 180,E1 30717.729,E2 30717.729} C_VEL
LIN {X 0,Y 644.65,Z 1075.667,A -85,B 0,C 180,E1 30715.688,E2 30715.688} C_VEL
LIN {X 0,Y 643.345,Z 1092.66,A -85,B 0,C 180,E1 30713.542,E2 30713.542} C_VEL
LIN {X 0,Y 642.443,Z 1106.088,A -85,B 0,C 180,E1 30711.645,E2 30711.645} C_VEL
LIN {X 0,Y 641.616,Z 1120.327,A -85,B 0,C 180,E1 30709.386,E2 30709.386} C_VEL
LIN {X 0,Y 640.946,Z 1132.926,A -85,B 0,C 180,E1 30707.054,E2 30707.054} C_VEL
LIN {X 0,Y 640.559,Z 1142.111,A -85,B 0,C 180,E1 30705.11,E2 30705.11} C_VEL
LIN {X 0,Y 640.289,Z 1150.404,A -85,B 0,C 180,E1 30703.087,E2 30703.087} C_VEL
LIN {X 0,Y 640.077,Z 1158.333,A -85,B 0,C 180,E1 30700.804,E2 30700.804} C_VEL
LIN {X 0,Y 639.985,Z 1165.018,A -85,B 0,C 180,E1 30698.354,E2 30698.354} C_VEL
LIN {X 0,Y 639.936,Z 1169.643,A -85,B 0,C 180,E1 30696.099,E2 30696.099} C_VEL
LIN {X 0,Y 639.913,Z 1172.941,A -85,B 0,C 180,E1 30693.763,E2 30693.763} C_VEL
LIN {X 0,Y 639.909,Z 1174.635,A -85,B 0,C 180,E1 30691.433,E2 30691.433} C_VEL
LIN {X 0,Y 639.894,Z 1174.861,A -85,B 0,C 180,E1 30689.373,E2 30689.373} C_VEL
LIN {X 0,Y 639.908,Z 1173.976,A -85,B 0,C 180,E1 30687.313,E2 30687.313} C_VEL
LIN {X 0,Y 639.919,Z 1171.616,A -85,B 0,C 180,E1 30685.07,E2 30685.07} C_VEL
LIN {X 0,Y 639.952,Z 1167.445,A -85,B 0,C 180,E1 30682.639,E2 30682.639} C_VEL
LIN {X 0,Y 640.024,Z 1161.75,A -85,B 0,C 180,E1 30680.287,E2 30680.287} C_VEL
LIN {X 0,Y 640.166,Z 1154.741,A -85,B 0,C 180,E1 30678.011,E2 30678.011} C_VEL
LIN {X 0,Y 640.476,Z 1144.939,A -85,B 0,C 180,E1 30675.443,E2 30675.443} C_VEL
LIN {X 0,Y 640.857,Z 1134.761,A -85,B 0,C 180,E1 30673.224,E2 30673.224} C_VEL
LIN {X 0,Y 641.356,Z 1124.485,A -85,B 0,C 180,E1 30671.268,E2 30671.268} C_VEL
LIN {X 0,Y 642.065,Z 1112.221,A -85,B 0,C 180,E1 30669.203,E2 30669.203} C_VEL
LIN {X 0,Y 643.1,Z 1096.126,A -85,B 0,C 180,E1 30666.837,E2 30666.837} C_VEL
LIN {X 0,Y 644.179,Z 1081.44,A -85,B 0,C 180,E1 30664.929,E2 30664.929} C_VEL
LIN {X 0,Y 645.644,Z 1063.26,A -85,B 0,C 180,E1 30662.816,E2 30662.816} C_VEL
LIN {X 0,Y 647.253,Z 1044.267,A -85,B 0,C 180,E1 30660.883,E2 30660.883} C_VEL
LIN {X 0,Y 648.705,Z 1027.882,A -85,B 0,C 180,E1 30659.376,E2 30659.376} C_VEL
LIN {X 0,Y 650.357,Z 1009.722,A -85,B 0,C 180,E1 30657.864,E2 30657.864} C_VEL
LIN {X 0,Y 652.486,Z 985.817,A -85,B 0,C 180,E1 30656.097,E2 30656.097} C_VEL
LIN {X 0,Y 654.312,Z 965.326,A -85,B 0,C 180,E1 30654.77,E2 30654.77} C_VEL
LIN {X 0,Y 656.117,Z 944.579,A -85,B 0,C 180,E1 30653.577,E2 30653.577} C_VEL
LIN {X 0,Y 658.216,Z 919.657,A -85,B 0,C 180,E1 30652.321,E2 30652.321} C_VEL
LIN {X 0,Y 660.017,Z 894.926,A -85,B 0,C 180,E1 30651.27,E2 30651.27} C_VEL
LIN {X 0,Y 661.393,Z 873.845,A -85,B 0,C 180,E1 30650.501,E2 30650.501} C_VEL
LIN {X 0,Y 662.73,Z 851.718,A -85,B 0,C 180,E1 30649.819,E2 30649.819} C_VEL
LIN {X 0,Y 664.085,Z 825.754,A -85,B 0,C 180,E1 30649.174,E2 30649.174} C_VEL
LIN {X 0,Y 665.082,Z 798.546,A -85,B 0,C 180,E1 30648.677,E2 30648.677} C_VEL
LIN {X 0,Y 667.462,Z 659.518,A -85,B 0,C 180,E1 30646.849,E2 30646.849} C_VEL
LIN {X 0,Y 671.142,Z 443.237,A -85,B 0,C 180,E1 30643.969,E2 30643.969} C_VEL
LIN {X 0,Y 672.346,Z 368.876,A -85,B 0,C 180,E1 30642.946,E2 30642.946} C_VEL
LIN {X 0,Y 662.934,Z 355.057,A -85,B 0,C 180,E1 30641.839,E2 30641.839} C_VEL
LIN {X 0,Y 652.285,Z 340.728,A -85,B 0,C 180,E1 30640.538,E2 30640.538} C_VEL
LIN {X 0,Y 649.001,Z 336.215,A -85,B 0,C 180,E1 30640.12,E2 30640.12} C_VEL
LIN {X 0,Y 645.628,Z 332.161,A -85,B 0,C 180,E1 30639.691,E2 30639.691} C_VEL
LIN {X 0,Y 644.618,Z 330.259,A -85,B 0,C 180,E1 30639.55,E2 30639.55} C_VEL
LIN {X 0,Y 641.94,Z 327.682,A -85,B 0,C 180,E1 30639.212,E2 30639.212} C_VEL
LIN {X 0,Y 640.779,Z 324.614,A -85,B 0,C 180,E1 30639.03,E2 30639.03} C_VEL
LIN {X 0,Y 640.727,Z 324.42,A -85,B 0,C 180,E1 30636.482,E2 30636.482} C_VEL
LIN {X 0,Y 640.799,Z 324.391,A -85,B 0,C 180,E1 30633.53,E2 30633.53} C_VEL
LIN {X 0,Y 640.724,Z 324.388,A -85,B 0,C 180,E1 30630.526,E2 30630.526} C_VEL
LIN {X 0,Y 640.745,Z 324.416,A -85,B 0,C 180,E1 30627.915,E2 30627.915} C_VEL
LIN {X 0,Y 640.747,Z 324.397,A -85,B 0,C 180,E1 30624.624,E2 30624.624} C_VEL
LIN {X 0,Y 640.738,Z 324.413,A -85,B 0,C 180,E1 30621.995,E2 30621.995} C_VEL
LIN {X 0,Y 640.814,Z 324.391,A -85,B 0,C 180,E1 30618.997,E2 30618.997} C_VEL
LIN {X 0,Y 640.742,Z 324.404,A -85,B 0,C 180,E1 30616.127,E2 30616.127} C_VEL
LIN {X 0,Y 640.771,Z 324.393,A -85,B 0,C 180,E1 30613.445,E2 30613.445} C_VEL
LIN {X 0,Y 640.759,Z 324.398,A -85,B 0,C 180,E1 30610.247,E2 30610.247} C_VEL
LIN {X 0,Y 640.76,Z 324.395,A -85,B 0,C 180,E1 30607.532,E2 30607.532} C_VEL
LIN {X 0,Y 640.792,Z 324.395,A -85,B 0,C 180,E1 30604.385,E2 30604.385} C_VEL
LIN {X 0,Y 640.757,Z 324.393,A -85,B 0,C 180,E1 30601.61,E2 30601.61} C_VEL
LIN {X 0,Y 640.833,Z 324.396,A -85,B 0,C 180,E1 30598.659,E2 30598.659} C_VEL
LIN {X 0,Y 640.762,Z 324.392,A -85,B 0,C 180,E1 30595.615,E2 30595.615} C_VEL
LIN {X 0,Y 640.835,Z 324.396,A -85,B 0,C 180,E1 30592.649,E2 30592.649} C_VEL
LIN {X 0,Y 640.771,Z 324.395,A -85,B 0,C 180,E1 30589.571,E2 30589.571} C_VEL
LIN {X 0,Y 640.823,Z 324.394,A -85,B 0,C 180,E1 30586.648,E2 30586.648} C_VEL
LIN {X 0,Y 640.781,Z 324.402,A -85,B 0,C 180,E1 30583.501,E2 30583.501} C_VEL
LIN {X 0,Y 640.816,Z 324.384,A -85,B 0,C 180,E1 30580.588,E2 30580.588} C_VEL
LIN {X 0,Y 640.789,Z 324.408,A -85,B 0,C 180,E1 30577.427,E2 30577.427} C_VEL
LIN {X 0,Y 640.824,Z 324.38,A -85,B 0,C 180,E1 30574.392,E2 30574.392} C_VEL
LIN {X 0,Y 640.793,Z 324.397,A -85,B 0,C 180,E1 30571.272,E2 30571.272} C_VEL
LIN {X 0,Y 640.829,Z 324.409,A -85,B 0,C 180,E1 30568.248,E2 30568.248} C_VEL
LIN {X 0,Y 640.796,Z 324.397,A -85,B 0,C 180,E1 30565.064,E2 30565.064} C_VEL
LIN {X 0,Y 640.814,Z 324.485,A -85,B 0,C 180,E1 30563.139,E2 30563.139} C_VEL
LIN {X 0,Y 642.001,Z 327.722,A -85,B 0,C 180,E1 30562.71,E2 30562.71} C_VEL
LIN {X 0,Y 643.089,Z 329.286,A -85,B 0,C 180,E1 30562.447,E2 30562.447} C_VEL
LIN {X 0,Y 644.952,Z 333.125,A -85,B 0,C 180,E1 30561.9,E2 30561.9} C_VEL
LIN {X 0,Y 653.191,Z 350.057,A -85,B 0,C 180,E1 30559.631,E2 30559.631} C_VEL
LIN {X 0,Y 671.003,Z 375.963,A -85,B 0,C 180,E1 30557.485,E2 30557.485} C_VEL
LIN {X 0,Y 672.754,Z 383.724,A -85,B 0,C 180,E1 30557.205,E2 30557.205} C_VEL
LIN {X 0,Y 669.102,Z 590.624,A -85,B 0,C 180,E1 30554.413,E2 30554.413} C_VEL
LIN {X 0,Y 665.489,Z 813.112,A -85,B 0,C 180,E1 30551.496,E2 30551.496} C_VEL
LIN {X 0,Y 664.62,Z 841.711,A -85,B 0,C 180,E1 30551.057,E2 30551.057} C_VEL
LIN {X 0,Y 663.6,Z 865.096,A -85,B 0,C 180,E1 30550.564,E2 30550.564} C_VEL
LIN {X 0,Y 662.356,Z 888.658,A -85,B 0,C 180,E1 30549.937,E2 30549.937} C_VEL
LIN {X 0,Y 660.608,Z 916.18,A -85,B 0,C 180,E1 30549.023,E2 30549.023} C_VEL
LIN {X 0,Y 658.904,Z 939.481,A -85,B 0,C 180,E1 30548.086,E2 30548.086} C_VEL
LIN {X 0,Y 657.248,Z 960.719,A -85,B 0,C 180,E1 30547.098,E2 30547.098} C_VEL
LIN {X 0,Y 655.353,Z 983.913,A -85,B 0,C 180,E1 30545.864,E2 30545.864} C_VEL
LIN {X 0,Y 653.233,Z 1007.869,A -85,B 0,C 180,E1 30544.388,E2 30544.388} C_VEL
LIN {X 0,Y 651.511,Z 1026.782,A -85,B 0,C 180,E1 30543.074,E2 30543.074} C_VEL
LIN {X 0,Y 649.826,Z 1045.274,A -85,B 0,C 180,E1 30541.647,E2 30541.647} C_VEL
LIN {X 0,Y 647.924,Z 1066.712,A -85,B 0,C 180,E1 30539.795,E2 30539.795} C_VEL
LIN {X 0,Y 646.294,Z 1085.553,A -85,B 0,C 180,E1 30537.944,E2 30537.944} C_VEL
LIN {X 0,Y 644.958,Z 1101.386,A -85,B 0,C 180,E1 30536.22,E2 30536.22} C_VEL
LIN {X 0,Y 643.6,Z 1119.538,A -85,B 0,C 180,E1 30534.004,E2 30534.004} C_VEL
LIN {X 0,Y 642.544,Z 1134.472,A -85,B 0,C 180,E1 30531.929,E2 30531.929} C_VEL
LIN {X 0,Y 641.755,Z 1147.161,A -85,B 0,C 180,E1 30529.95,E2 30529.95} C_VEL
LIN {X 0,Y 641.061,Z 1160.82,A -85,B 0,C 180,E1 30527.519,E2 30527.519} C_VEL
LIN {X 0,Y 640.585,Z 1171.078,A -85,B 0,C 180,E1 30525.387,E2 30525.387} C_VEL
LIN {X 0,Y 640.329,Z 1179.159,A -85,B 0,C 180,E1 30523.454,E2 30523.454} C_VEL
LIN {X 0,Y 640.122,Z 1186.713,A -85,B 0,C 180,E1 30521.35,E2 30521.35} C_VEL
LIN {X 0,Y 639.995,Z 1193.595,A -85,B 0,C 180,E1 30518.988,E2 30518.988} C_VEL
LIN {X 0,Y 639.937,Z 1198.925,A -85,B 0,C 180,E1 30516.549,E2 30516.549} C_VEL
LIN {X 0,Y 639.918,Z 1202.36,A -85,B 0,C 180,E1 30514.301,E2 30514.301} C_VEL
LIN {X 0,Y 639.909,Z 1204.494,A -85,B 0,C 180,E1 30511.88,E2 30511.88} C_VEL
LIN {X 0,Y 639.892,Z 1204.872,A -85,B 0,C 180,E1 30509.463,E2 30509.463} C_VEL
LIN {X 0,Y 639.91,Z 1203.941,A -85,B 0,C 180,E1 30507.313,E2 30507.313} C_VEL
LIN {X 0,Y 639.922,Z 1201.552,A -85,B 0,C 180,E1 30505.07,E2 30505.07} C_VEL
LIN {X 0,Y 639.953,Z 1197.347,A -85,B 0,C 180,E1 30502.639,E2 30502.639} C_VEL
LIN {X 0,Y 640.026,Z 1191.624,A -85,B 0,C 180,E1 30500.287,E2 30500.287} C_VEL
LIN {X 0,Y 640.164,Z 1184.591,A -85,B 0,C 180,E1 30498.011,E2 30498.011} C_VEL
LIN {X 0,Y 640.484,Z 1174.741,A -85,B 0,C 180,E1 30495.443,E2 30495.443} C_VEL
LIN {X 0,Y 640.843,Z 1165.001,A -85,B 0,C 180,E1 30493.317,E2 30493.317} C_VEL
LIN {X 0,Y 641.352,Z 1154.761,A -85,B 0,C 180,E1 30491.362,E2 30491.362} C_VEL
LIN {X 0,Y 642.053,Z 1142.531,A -85,B 0,C 180,E1 30489.298,E2 30489.298} C_VEL
LIN {X 0,Y 643.082,Z 1126.501,A -85,B 0,C 180,E1 30486.933,E2 30486.933} C_VEL
LIN {X 0,Y 644.144,Z 1111.859,A -85,B 0,C 180,E1 30485.026,E2 30485.026} C_VEL
LIN {X 0,Y 645.467,Z 1095.435,A -85,B 0,C 180,E1 30483.107,E2 30483.107} C_VEL
LIN {X 0,Y 647.156,Z 1075.337,A -85,B 0,C 180,E1 30481.03,E2 30481.03} C_VEL
LIN {X 0,Y 648.61,Z 1058.942,A -85,B 0,C 180,E1 30479.514,E2 30479.514} C_VEL
LIN {X 0,Y 650.17,Z 1041.626,A -85,B 0,C 180,E1 30478.061,E2 30478.061} C_VEL
LIN {X 0,Y 652.2,Z 1019.55,A -85,B 0,C 180,E1 30476.397,E2 30476.397} C_VEL
LIN {X 0,Y 654.232,Z 996.179,A -85,B 0,C 180,E1 30474.867,E2 30474.867} C_VEL
LIN {X 0,Y 655.998,Z 975.858,A -85,B 0,C 180,E1 30473.691,E2 30473.691} C_VEL
LIN {X 0,Y 657.988,Z 952.264,A -85,B 0,C 180,E1 30472.49,E2 30472.49} C_VEL
LIN {X 0,Y 659.917,Z 926.451,A -85,B 0,C 180,E1 30471.374,E2 30471.374} C_VEL
LIN {X 0,Y 661.328,Z 904.877,A -85,B 0,C 180,E1 30470.58,E2 30470.58} C_VEL
LIN {X 0,Y 662.652,Z 883.014,A -85,B 0,C 180,E1 30469.901,E2 30469.901} C_VEL
LIN {X 0,Y 663.947,Z 858.262,A -85,B 0,C 180,E1 30469.275,E2 30469.275} C_VEL
LIN {X 0,Y 665.053,Z 829.748,A -85,B 0,C 180,E1 30468.74,E2 30468.74} C_VEL
LIN {X 0,Y 666.538,Z 746.821,A -85,B 0,C 180,E1 30467.643,E2 30467.643} C_VEL
LIN {X 0,Y 670.249,Z 524.284,A -85,B 0,C 180,E1 30464.702,E2 30464.702} C_VEL
LIN {X 0,Y 672.655,Z 382.626,A -85,B 0,C 180,E1 30462.769,E2 30462.769} C_VEL
LIN {X 0,Y 670.78,Z 375.624,A -85,B 0,C 180,E1 30462.489,E2 30462.489} C_VEL
LIN {X 0,Y 655.84,Z 354.031,A -85,B 0,C 180,E1 30460.704,E2 30460.704} C_VEL
LIN {X 0,Y 652.611,Z 349.14,A -85,B 0,C 180,E1 30460.273,E2 30460.273} C_VEL
LIN {X 0,Y 646.459,Z 336.509,A -85,B 0,C 180,E1 30458.56,E2 30458.56} C_VEL
LIN {X 0,Y 644.482,Z 332.461,A -85,B 0,C 180,E1 30457.99,E2 30457.99} C_VEL
LIN {X 0,Y 642.753,Z 328.702,A -85,B 0,C 180,E1 30457.464,E2 30457.464} C_VEL
LIN {X 0,Y 641.091,Z 325.767,A -85,B 0,C 180,E1 30457.011,E2 30457.011} C_VEL
LIN {X 0,Y 640.804,Z 324.388,A -85,B 0,C 180,E1 30456.812,E2 30456.812} C_VEL
LIN {X 0,Y 640.818,Z 324.381,A -85,B 0,C 180,E1 30453.636,E2 30453.636} C_VEL
LIN {X 0,Y 640.813,Z 324.387,A -85,B 0,C 180,E1 30450.539,E2 30450.539} C_VEL
LIN {X 0,Y 640.802,Z 324.408,A -85,B 0,C 180,E1 30447.307,E2 30447.307} C_VEL
LIN {X 0,Y 640.822,Z 324.388,A -85,B 0,C 180,E1 30444.228,E2 30444.228} C_VEL
LIN {X 0,Y 640.789,Z 324.386,A -85,B 0,C 180,E1 30441.078,E2 30441.078} C_VEL
LIN {X 0,Y 640.818,Z 324.402,A -85,B 0,C 180,E1 30438.09,E2 30438.09} C_VEL
LIN {X 0,Y 640.781,Z 324.38,A -85,B 0,C 180,E1 30434.92,E2 30434.92} C_VEL
LIN {X 0,Y 640.814,Z 324.406,A -85,B 0,C 180,E1 30431.958,E2 30431.958} C_VEL
LIN {X 0,Y 640.777,Z 324.382,A -85,B 0,C 180,E1 30428.796,E2 30428.796} C_VEL
LIN {X 0,Y 640.79,Z 324.408,A -85,B 0,C 180,E1 30426.001,E2 30426.001} C_VEL
LIN {X 0,Y 640.78,Z 324.381,A -85,B 0,C 180,E1 30422.773,E2 30422.773} C_VEL
LIN {X 0,Y 640.773,Z 324.409,A -85,B 0,C 180,E1 30420,E2 30420} C_VEL
LIN {X 0,Y 640.798,Z 324.378,A -85,B 0,C 180,E1 30416.869,E2 30416.869} C_VEL
LIN {X 0,Y 640.759,Z 324.411,A -85,B 0,C 180,E1 30414.089,E2 30414.089} C_VEL
LIN {X 0,Y 640.83,Z 324.375,A -85,B 0,C 180,E1 30411.114,E2 30411.114} C_VEL
LIN {X 0,Y 640.753,Z 324.413,A -85,B 0,C 180,E1 30408.113,E2 30408.113} C_VEL
LIN {X 0,Y 640.798,Z 324.379,A -85,B 0,C 180,E1 30405.265,E2 30405.265} C_VEL
LIN {X 0,Y 640.753,Z 324.413,A -85,B 0,C 180,E1 30402.151,E2 30402.151} C_VEL
LIN {X 0,Y 640.75,Z 324.382,A -85,B 0,C 180,E1 30399.54,E2 30399.54} C_VEL
LIN {X 0,Y 640.79,Z 324.408,A -85,B 0,C 180,E1 30396.455,E2 30396.455} C_VEL
LIN {X 0,Y 640.736,Z 324.394,A -85,B 0,C 180,E1 30393.692,E2 30393.692} C_VEL
LIN {X 0,Y 640.796,Z 324.397,A -85,B 0,C 180,E1 30390.867,E2 30390.867} C_VEL
LIN {X 0,Y 640.742,Z 324.418,A -85,B 0,C 180,E1 30387.85,E2 30387.85} C_VEL
LIN {X 0,Y 640.738,Z 324.388,A -85,B 0,C 180,E1 30385.166,E2 30385.166} C_VEL
LIN {X 0,Y 640.755,Z 324.389,A -85,B 0,C 180,E1 30382.001,E2 30382.001} C_VEL
LIN {X 0,Y 640.767,Z 324.526,A -85,B 0,C 180,E1 30380.882,E2 30380.882} C_VEL
LIN {X 0,Y 641.924,Z 327.642,A -85,B 0,C 180,E1 30380.7,E2 30380.7} C_VEL
LIN {X 0,Y 644.599,Z 330.246,A -85,B 0,C 180,E1 30380.363,E2 30380.363} C_VEL
LIN {X 0,Y 647.373,Z 334.587,A -85,B 0,C 180,E1 30379.99,E2 30379.99} C_VEL
LIN {X 0,Y 649.327,Z 336.816,A -85,B 0,C 180,E1 30379.746,E2 30379.746} C_VEL
LIN {X 0,Y 652.714,Z 341.143,A -85,B 0,C 180,E1 30379.321,E2 30379.321} C_VEL
LIN {X 0,Y 666.321,Z 359.8,A -85,B 0,C 180,E1 30377.67,E2 30377.67} C_VEL
LIN {X 0,Y 669.837,Z 365.18,A -85,B 0,C 180,E1 30377.254,E2 30377.254} C_VEL
LIN {X 0,Y 670.691,Z 368.173,A -85,B 0,C 180,E1 30377.128,E2 30377.128} C_VEL
LIN {X 0,Y 670.436,Z 372.482,A -85,B 0,C 180,E1 30377.085,E2 30377.085} C_VEL
LIN {X 0,Y 666.977,Z 385.695,A -85,B 0,C 180,E1 30377.202,E2 30377.202} C_VEL
LIN {X 0,Y 666.647,Z 388.952,A -85,B 0,C 180,E1 30377.182,E2 30377.182} C_VEL
LIN {X 0,Y 662.44,Z 613.036,A -85,B 0,C 180,E1 30374.154,E2 30374.154} C_VEL
LIN {X 0,Y 659.082,Z 797.759,A -85,B 0,C 180,E1 30371.705,E2 30371.705} C_VEL
LIN {X 0,Y 658.058,Z 824.543,A -85,B 0,C 180,E1 30371.222,E2 30371.222} C_VEL
LIN {X 0,Y 656.594,Z 851.134,A -85,B 0,C 180,E1 30370.563,E2 30370.563} C_VEL
LIN {X 0,Y 655.197,Z 872.967,A -85,B 0,C 180,E1 30369.89,E2 30369.89} C_VEL
LIN {X 0,Y 653.71,Z 894.017,A -85,B 0,C 180,E1 30369.124,E2 30369.124} C_VEL
LIN {X 0,Y 651.951,Z 916.467,A -85,B 0,C 180,E1 30368.174,E2 30368.174} C_VEL
LIN {X 0,Y 649.699,Z 942.42,A -85,B 0,C 180,E1 30366.884,E2 30366.884} C_VEL
LIN {X 0,Y 647.761,Z 963.154,A -85,B 0,C 180,E1 30365.695,E2 30365.695} C_VEL
LIN {X 0,Y 645.924,Z 982.388,A -85,B 0,C 180,E1 30364.456,E2 30364.456} C_VEL
LIN {X 0,Y 643.846,Z 1003.651,A -85,B 0,C 180,E1 30362.924,E2 30362.924} C_VEL
LIN {X 0,Y 641.689,Z 1025.805,A -85,B 0,C 180,E1 30361.1,E2 30361.1} C_VEL
LIN {X 0,Y 640.108,Z 1042.359,A -85,B 0,C 180,E1 30359.577,E2 30359.577} C_VEL
LIN {X 0,Y 638.581,Z 1058.754,A -85,B 0,C 180,E1 30357.915,E2 30357.915} C_VEL
LIN {X 0,Y 636.858,Z 1078.392,A -85,B 0,C 180,E1 30355.678,E2 30355.678} C_VEL
LIN {X 0,Y 635.603,Z 1093.622,A -85,B 0,C 180,E1 30353.713,E2 30353.713} C_VEL
LIN {X 0,Y 634.603,Z 1107.36,A -85,B 0,C 180,E1 30351.731,E2 30351.731} C_VEL
LIN {X 0,Y 633.644,Z 1122.427,A -85,B 0,C 180,E1 30349.256,E2 30349.256} C_VEL
LIN {X 0,Y 633.017,Z 1133.642,A -85,B 0,C 180,E1 30347.129,E2 30347.129} C_VEL
LIN {X 0,Y 632.596,Z 1142.927,A -85,B 0,C 180,E1 30345.117,E2 30345.117} C_VEL
LIN {X 0,Y 632.274,Z 1152.523,A -85,B 0,C 180,E1 30342.698,E2 30342.698} C_VEL
LIN {X 0,Y 632.069,Z 1160.479,A -85,B 0,C 180,E1 30340.205,E2 30340.205} C_VEL
LIN {X 0,Y 631.973,Z 1166.255,A -85,B 0,C 180,E1 30337.912,E2 30337.912} C_VEL
LIN {X 0,Y 631.923,Z 1170.857,A -85,B 0,C 180,E1 30335.448,E2 30335.448} C_VEL
LIN {X 0,Y 631.912,Z 1173.701,A -85,B 0,C 180,E1 30332.993,E2 30332.993} C_VEL
LIN {X 0,Y 631.905,Z 1174.771,A -85,B 0,C 180,E1 30330.907,E2 30330.907} C_VEL
LIN {X 0,Y 631.908,Z 1174.771,A -85,B 0,C 180,E1 30329.003,E2 30329.003} C_VEL
LIN {X 0,Y 631.914,Z 1173.7,A -85,B 0,C 180,E1 30326.916,E2 30326.916} C_VEL
LIN {X 0,Y 631.922,Z 1170.856,A -85,B 0,C 180,E1 30324.461,E2 30324.461} C_VEL
LIN {X 0,Y 631.973,Z 1166.252,A -85,B 0,C 180,E1 30321.997,E2 30321.997} C_VEL
LIN {X 0,Y 632.068,Z 1160.474,A -85,B 0,C 180,E1 30319.703,E2 30319.703} C_VEL
LIN {X 0,Y 632.276,Z 1152.514,A -85,B 0,C 180,E1 30317.209,E2 30317.209} C_VEL
LIN {X 0,Y 632.579,Z 1143.315,A -85,B 0,C 180,E1 30314.883,E2 30314.883} C_VEL
LIN {X 0,Y 633.011,Z 1133.835,A -85,B 0,C 180,E1 30312.82,E2 30312.82} C_VEL
LIN {X 0,Y 633.614,Z 1122.915,A -85,B 0,C 180,E1 30310.743,E2 30310.743} C_VEL
LIN {X 0,Y 634.563,Z 1107.946,A -85,B 0,C 180,E1 30308.267,E2 30308.267} C_VEL
LIN {X 0,Y 635.571,Z 1094.017,A -85,B 0,C 180,E1 30306.251,E2 30306.251} C_VEL
LIN {X 0,Y 636.797,Z 1079.096,A -85,B 0,C 180,E1 30304.319,E2 30304.319} C_VEL
LIN {X 0,Y 638.502,Z 1059.574,A -85,B 0,C 180,E1 30302.081,E2 30302.081} C_VEL
LIN {X 0,Y 640.071,Z 1042.738,A -85,B 0,C 180,E1 30300.37,E2 30300.37} C_VEL
LIN {X 0,Y 641.683,Z 1025.828,A -85,B 0,C 180,E1 30298.812,E2 30298.812} C_VEL
LIN {X 0,Y 643.836,Z 1003.794,A -85,B 0,C 180,E1 30296.996,E2 30296.996} C_VEL
LIN {X 0,Y 645.876,Z 982.889,A -85,B 0,C 180,E1 30295.487,E2 30295.487} C_VEL
LIN {X 0,Y 647.711,Z 963.688,A -85,B 0,C 180,E1 30294.248,E2 30294.248} C_VEL
LIN {X 0,Y 649.644,Z 942.988,A -85,B 0,C 180,E1 30293.058,E2 30293.058} C_VEL
LIN {X 0,Y 651.824,Z 918.263,A -85,B 0,C 180,E1 30291.817,E2 30291.817} C_VEL
LIN {X 0,Y 653.651,Z 894.906,A -85,B 0,C 180,E1 30290.821,E2 30290.821} C_VEL
LIN {X 0,Y 655.135,Z 873.823,A -85,B 0,C 180,E1 30290.048,E2 30290.048} C_VEL
LIN {X 0,Y 656.554,Z 851.788,A -85,B 0,C 180,E1 30289.366,E2 30289.366} C_VEL
LIN {X 0,Y 657.981,Z 826.134,A -85,B 0,C 180,E1 30288.724,E2 30288.724} C_VEL
LIN {X 0,Y 659.055,Z 798.792,A -85,B 0,C 180,E1 30288.22,E2 30288.22} C_VEL
LIN {X 0,Y 661.041,Z 692.432,A -85,B 0,C 180,E1 30286.808,E2 30286.808} C_VEL
LIN {X 0,Y 664.946,Z 476.624,A -85,B 0,C 180,E1 30283.925,E2 30283.925} C_VEL
LIN {X 0,Y 666.84,Z 372.768,A -85,B 0,C 180,E1 30282.493,E2 30282.493} C_VEL
LIN {X 0,Y 658.757,Z 360.875,A -85,B 0,C 180,E1 30281.523,E2 30281.523} C_VEL
LIN {X 0,Y 648.471,Z 346.998,A -85,B 0,C 180,E1 30280.246,E2 30280.246} C_VEL
LIN {X 0,Y 644.047,Z 341.325,A -85,B 0,C 180,E1 30279.678,E2 30279.678} C_VEL
LIN {X 0,Y 640.4,Z 336.42,A -85,B 0,C 180,E1 30279.195,E2 30279.195} C_VEL
LIN {X 0,Y 637.538,Z 332.751,A -85,B 0,C 180,E1 30278.811,E2 30278.811} C_VEL
LIN {X 0,Y 636.664,Z 331.308,A -85,B 0,C 180,E1 30278.687,E2 30278.687} C_VEL
LIN {X 0,Y 634.038,Z 328.799,A -85,B 0,C 180,E1 30278.343,E2 30278.343} C_VEL
LIN {X 0,Y 632.838,Z 325.653,A -85,B 0,C 180,E1 30278.147,E2 30278.147} C_VEL
LIN {X 0,Y 632.865,Z 325.375,A -85,B 0,C 180,E1 30275.439,E2 30275.439} C_VEL
LIN {X 0,Y 632.785,Z 325.408,A -85,B 0,C 180,E1 30272.46,E2 30272.46} C_VEL
LIN {X 0,Y 632.833,Z 325.373,A -85,B 0,C 180,E1 30269.64,E2 30269.64} C_VEL
LIN {X 0,Y 632.798,Z 325.388,A -85,B 0,C 180,E1 30266.562,E2 30266.562} C_VEL
LIN {X 0,Y 632.807,Z 325.396,A -85,B 0,C 180,E1 30263.86,E2 30263.86} C_VEL
LIN {X 0,Y 632.819,Z 325.368,A -85,B 0,C 180,E1 30260.631,E2 30260.631} C_VEL
LIN {X 0,Y 632.804,Z 325.402,A -85,B 0,C 180,E1 30257.946,E2 30257.946} C_VEL
LIN {X 0,Y 632.884,Z 325.362,A -85,B 0,C 180,E1 30254.923,E2 30254.923} C_VEL
LIN {X 0,Y 632.809,Z 325.402,A -85,B 0,C 180,E1 30251.946,E2 30251.946} C_VEL
LIN {X 0,Y 632.879,Z 325.362,A -85,B 0,C 180,E1 30248.999,E2 30248.999} C_VEL
LIN {X 0,Y 632.817,Z 325.401,A -85,B 0,C 180,E1 30245.986,E2 30245.986} C_VEL
LIN {X 0,Y 632.847,Z 325.367,A -85,B 0,C 180,E1 30243.17,E2 30243.17} C_VEL
LIN {X 0,Y 632.832,Z 325.399,A -85,B 0,C 180,E1 30240,E2 30240} C_VEL
LIN {X 0,Y 632.838,Z 325.37,A -85,B 0,C 180,E1 30237.192,E2 30237.192} C_VEL
LIN {X 0,Y 632.843,Z 325.397,A -85,B 0,C 180,E1 30233.923,E2 30233.923} C_VEL
LIN {X 0,Y 632.841,Z 325.369,A -85,B 0,C 180,E1 30231.092,E2 30231.092} C_VEL
LIN {X 0,Y 632.856,Z 325.396,A -85,B 0,C 180,E1 30227.87,E2 30227.87} C_VEL
LIN {X 0,Y 632.844,Z 325.367,A -85,B 0,C 180,E1 30224.982,E2 30224.982} C_VEL
LIN {X 0,Y 632.865,Z 325.393,A -85,B 0,C 180,E1 30221.77,E2 30221.77} C_VEL
LIN {X 0,Y 632.858,Z 325.374,A -85,B 0,C 180,E1 30218.771,E2 30218.771} C_VEL
LIN {X 0,Y 632.858,Z 325.376,A -85,B 0,C 180,E1 30215.509,E2 30215.509} C_VEL
LIN {X 0,Y 632.885,Z 325.4,A -85,B 0,C 180,E1 30212.425,E2 30212.425} C_VEL
LIN {X 0,Y 632.854,Z 325.382,A -85,B 0,C 180,E1 30209.209,E2 30209.209} C_VEL
LIN {X 0,Y 632.885,Z 325.367,A -85,B 0,C 180,E1 30206.201,E2 30206.201} C_VEL
LIN {X 0,Y 632.92,Z 325.622,A -85,B 0,C 180,E1 30203.956,E2 30203.956} C_VEL
LIN {X 0,Y 634.104,Z 328.729,A -85,B 0,C 180,E1 30203.525,E2 30203.525} C_VEL
LIN {X 0,Y 635.184,Z 330.356,A -85,B 0,C 180,E1 30203.247,E2 30203.247} C_VEL
LIN {X 0,Y 636.958,Z 334.063,A -85,B 0,C 180,E1 30202.703,E2 30202.703} C_VEL
LIN {X 0,Y 643.898,Z 348.292,A -85,B 0,C 180,E1 30200.686,E2 30200.686} C_VEL
LIN {X 0,Y 645.451,Z 350.852,A -85,B 0,C 180,E1 30200.425,E2 30200.425} C_VEL
LIN {X 0,Y 659.318,Z 370.746,A -85,B 0,C 180,E1 30198.679,E2 30198.679} C_VEL
LIN {X 0,Y 666.315,Z 381.343,A -85,B 0,C 180,E1 30197.839,E2 30197.839} C_VEL
LIN {X 0,Y 667.249,Z 385.995,A -85,B 0,C 180,E1 30197.678,E2 30197.678} C_VEL
LIN {X 0,Y 663.35,Z 592.544,A -85,B 0,C 180,E1 30194.873,E2 30194.873} C_VEL
LIN {X 0,Y 659.46,Z 815.271,A -85,B 0,C 180,E1 30191.931,E2 30191.931} C_VEL
LIN {X 0,Y 658.528,Z 842.66,A -85,B 0,C 180,E1 30191.499,E2 30191.499} C_VEL
LIN {X 0,Y 657.461,Z 865.505,A -85,B 0,C 180,E1 30191.012,E2 30191.012} C_VEL
LIN {X 0,Y 656.135,Z 888.998,A -85,B 0,C 180,E1 30190.382,E2 30190.382} C_VEL
LIN {X 0,Y 654.293,Z 916.177,A -85,B 0,C 180,E1 30189.473,E2 30189.473} C_VEL
LIN {X 0,Y 652.464,Z 939.478,A -85,B 0,C 180,E1 30188.531,E2 30188.531} C_VEL
LIN {X 0,Y 650.698,Z 960.613,A -85,B 0,C 180,E1 30187.542,E2 30187.542} C_VEL
LIN {X 0,Y 648.609,Z 984.359,A -85,B 0,C 180,E1 30186.268,E2 30186.268} C_VEL
LIN {X 0,Y 646.316,Z 1008.463,A -85,B 0,C 180,E1 30184.765,E2 30184.765} C_VEL
LIN {X 0,Y 644.518,Z 1026.911,A -85,B 0,C 180,E1 30183.47,E2 30183.47} C_VEL
LIN {X 0,Y 642.774,Z 1044.668,A -85,B 0,C 180,E1 30182.087,E2 30182.087} C_VEL
LIN {X 0,Y 640.75,Z 1065.691,A -85,B 0,C 180,E1 30180.267,E2 30180.267} C_VEL
LIN {X 0,Y 638.927,Z 1084.996,A -85,B 0,C 180,E1 30178.356,E2 30178.356} C_VEL
LIN {X 0,Y 637.498,Z 1100.835,A -85,B 0,C 180,E1 30176.616,E2 30176.616} C_VEL
LIN {X 0,Y 636.015,Z 1118.728,A -85,B 0,C 180,E1 30174.422,E2 30174.422} C_VEL
LIN {X 0,Y 634.844,Z 1133.829,A -85,B 0,C 180,E1 30172.307,E2 30172.307} C_VEL
LIN {X 0,Y 633.985,Z 1146.586,A -85,B 0,C 180,E1 30170.302,E2 30170.302} C_VEL
LIN {X 0,Y 633.228,Z 1159.89,A -85,B 0,C 180,E1 30167.933,E2 30167.933} C_VEL
LIN {X 0,Y 632.659,Z 1171.079,A -85,B 0,C 180,E1 30165.585,E2 30165.585} C_VEL
LIN {X 0,Y 632.373,Z 1179.16,A -85,B 0,C 180,E1 30163.626,E2 30163.626} C_VEL
LIN {X 0,Y 632.151,Z 1186.71,A -85,B 0,C 180,E1 30161.495,E2 30161.495} C_VEL
LIN {X 0,Y 632.004,Z 1193.595,A -85,B 0,C 180,E1 30159.103,E2 30159.103} C_VEL
LIN {X 0,Y 631.938,Z 1198.922,A -85,B 0,C 180,E1 30156.633,E2 30156.633} C_VEL
LIN {X 0,Y 631.917,Z 1202.357,A -85,B 0,C 180,E1 30154.356,E2 30154.356} C_VEL
LIN {X 0,Y 631.911,Z 1204.438,A -85,B 0,C 180,E1 30151.995,E2 30151.995} C_VEL
LIN {X 0,Y 631.892,Z 1204.894,A -85,B 0,C 180,E1 30149.547,E2 30149.547} C_VEL
LIN {X 0,Y 631.909,Z 1204.007,A -85,B 0,C 180,E1 30147.37,E2 30147.37} C_VEL
LIN {X 0,Y 631.921,Z 1201.674,A -85,B 0,C 180,E1 30145.099,E2 30145.099} C_VEL
LIN {X 0,Y 631.956,Z 1197.542,A -85,B 0,C 180,E1 30142.637,E2 30142.637} C_VEL
LIN {X 0,Y 632.034,Z 1191.875,A -85,B 0,C 180,E1 30140.255,E2 30140.255} C_VEL
LIN {X 0,Y 632.182,Z 1184.891,A -85,B 0,C 180,E1 30137.95,E2 30137.95} C_VEL
LIN {X 0,Y 632.529,Z 1175.145,A -85,B 0,C 180,E1 30135.35,E2 30135.35} C_VEL
LIN {X 0,Y 632.943,Z 1165,A -85,B 0,C 180,E1 30133.102,E2 30133.102} C_VEL
LIN {X 0,Y 633.497,Z 1154.763,A -85,B 0,C 180,E1 30131.122,E2 30131.122} C_VEL
LIN {X 0,Y 634.299,Z 1141.95,A -85,B 0,C 180,E1 30128.937,E2 30128.937} C_VEL
LIN {X 0,Y 635.434,Z 1125.798,A -85,B 0,C 180,E1 30126.541,E2 30126.541} C_VEL
LIN {X 0,Y 636.63,Z 1111.083,A -85,B 0,C 180,E1 30124.611,E2 30124.611} C_VEL
LIN {X 0,Y 638.206,Z 1092.836,A -85,B 0,C 180,E1 30122.47,E2 30122.47} C_VEL
LIN {X 0,Y 639.969,Z 1073.816,A -85,B 0,C 180,E1 30120.519,E2 30120.519} C_VEL
LIN {X 0,Y 641.533,Z 1057.513,A -85,B 0,C 180,E1 30119.007,E2 30119.007} C_VEL
LIN {X 0,Y 643.319,Z 1039.19,A -85,B 0,C 180,E1 30117.469,E2 30117.469} C_VEL
LIN {X 0,Y 645.642,Z 1015.192,A -85,B 0,C 180,E1 30115.688,E2 30115.688} C_VEL
LIN {X 0,Y 647.617,Z 994.635,A -85,B 0,C 180,E1 30114.351,E2 30114.351} C_VEL
LIN {X 0,Y 649.503,Z 974.415,A -85,B 0,C 180,E1 30113.181,E2 30113.181} C_VEL
LIN {X 0,Y 651.753,Z 949.295,A -85,B 0,C 180,E1 30111.908,E2 30111.908} C_VEL
LIN {X 0,Y 653.674,Z 924.586,A -85,B 0,C 180,E1 30110.854,E2 30110.854} C_VEL
LIN {X 0,Y 655.115,Z 904.135,A -85,B 0,C 180,E1 30110.104,E2 30110.104} C_VEL
LIN {X 0,Y 656.512,Z 882.385,A -85,B 0,C 180,E1 30109.428,E2 30109.428} C_VEL
LIN {X 0,Y 657.909,Z 857.375,A -85,B 0,C 180,E1 30108.797,E2 30108.797} C_VEL
LIN {X 0,Y 659.043,Z 829.291,A -85,B 0,C 180,E1 30108.273,E2 30108.273} C_VEL
LIN {X 0,Y 660.722,Z 741.104,A -85,B 0,C 180,E1 30107.099,E2 30107.099} C_VEL
LIN {X 0,Y 664.731,Z 518.505,A -85,B 0,C 180,E1 30104.131,E2 30104.131} C_VEL
LIN {X 0,Y 667.154,Z 384.808,A -85,B 0,C 180,E1 30102.294,E2 30102.294} C_VEL
LIN {X 0,Y 665.874,Z 380.338,A -85,B 0,C 180,E1 30102.104,E2 30102.104} C_VEL
LIN {X 0,Y 651.417,Z 359.457,A -85,B 0,C 180,E1 30100.343,E2 30100.343} C_VEL
LIN {X 0,Y 644.074,Z 348.703,A -85,B 0,C 180,E1 30099.368,E2 30099.368} C_VEL
LIN {X 0,Y 638.466,Z 337.29,A -85,B 0,C 180,E1 30097.759,E2 30097.759} C_VEL
LIN {X 0,Y 636.592,Z 333.545,A -85,B 0,C 180,E1 30097.209,E2 30097.209} C_VEL
LIN {X 0,Y 634.452,Z 329.231,A -85,B 0,C 180,E1 30096.565,E2 30096.565} C_VEL
LIN {X 0,Y 633.005,Z 326.088,A -85,B 0,C 180,E1 30096.1,E2 30096.1} C_VEL
LIN {X 0,Y 632.887,Z 325.394,A -85,B 0,C 180,E1 30095.995,E2 30095.995} C_VEL
LIN {X 0,Y 632.853,Z 325.381,A -85,B 0,C 180,E1 30092.923,E2 30092.923} C_VEL
LIN {X 0,Y 632.888,Z 325.365,A -85,B 0,C 180,E1 30089.846,E2 30089.846} C_VEL
LIN {X 0,Y 632.849,Z 325.394,A -85,B 0,C 180,E1 30086.864,E2 30086.864} C_VEL
LIN {X 0,Y 632.891,Z 325.382,A -85,B 0,C 180,E1 30083.758,E2 30083.758} C_VEL
LIN {X 0,Y 632.841,Z 325.371,A -85,B 0,C 180,E1 30080.824,E2 30080.824} C_VEL
LIN {X 0,Y 632.893,Z 325.394,A -85,B 0,C 180,E1 30077.753,E2 30077.753} C_VEL
LIN {X 0,Y 632.836,Z 325.367,A -85,B 0,C 180,E1 30074.737,E2 30074.737} C_VEL
LIN {X 0,Y 632.891,Z 325.395,A -85,B 0,C 180,E1 30071.76,E2 30071.76} C_VEL
LIN {X 0,Y 632.832,Z 325.371,A -85,B 0,C 180,E1 30068.633,E2 30068.633} C_VEL
LIN {X 0,Y 632.881,Z 325.396,A -85,B 0,C 180,E1 30065.712,E2 30065.712} C_VEL
LIN {X 0,Y 632.831,Z 325.37,A -85,B 0,C 180,E1 30062.626,E2 30062.626} C_VEL
LIN {X 0,Y 632.849,Z 325.398,A -85,B 0,C 180,E1 30059.819,E2 30059.819} C_VEL
LIN {X 0,Y 632.836,Z 325.369,A -85,B 0,C 180,E1 30056.649,E2 30056.649} C_VEL
LIN {X 0,Y 632.831,Z 325.399,A -85,B 0,C 180,E1 30053.832,E2 30053.832} C_VEL
LIN {X 0,Y 632.842,Z 325.368,A -85,B 0,C 180,E1 30050.634,E2 30050.634} C_VEL
LIN {X 0,Y 632.816,Z 325.401,A -85,B 0,C 180,E1 30047.869,E2 30047.869} C_VEL
LIN {X 0,Y 632.877,Z 325.364,A -85,B 0,C 180,E1 30044.795,E2 30044.795} C_VEL
LIN {X 0,Y 632.809,Z 325.401,A -85,B 0,C 180,E1 30041.864,E2 30041.864} C_VEL
LIN {X 0,Y 632.885,Z 325.364,A -85,B 0,C 180,E1 30038.886,E2 30038.886} C_VEL
LIN {X 0,Y 632.805,Z 325.396,A -85,B 0,C 180,E1 30035.942,E2 30035.942} C_VEL
LIN {X 0,Y 632.822,Z 325.387,A -85,B 0,C 180,E1 30033.214,E2 30033.214} C_VEL
LIN {X 0,Y 632.805,Z 325.373,A -85,B 0,C 180,E1 30029.981,E2 30029.981} C_VEL
LIN {X 0,Y 632.796,Z 325.407,A -85,B 0,C 180,E1 30027.37,E2 30027.37} C_VEL
LIN {X 0,Y 632.853,Z 325.381,A -85,B 0,C 180,E1 30024.299,E2 30024.299} C_VEL
LIN {X 0,Y 632.828,Z 325.619,A -85,B 0,C 180,E1 30021.764,E2 30021.764} C_VEL
LIN {X 0,Y 634.019,Z 328.756,A -85,B 0,C 180,E1 30021.57,E2 30021.57} C_VEL
LIN {X 0,Y 636.499,Z 331.184,A -85,B 0,C 180,E1 30021.243,E2 30021.243} C_VEL
LIN {X 0,Y 637.456,Z 332.583,A -85,B 0,C 180,E1 30021.11,E2 30021.11} C_VEL
LIN {X 0,Y 640.239,Z 336.261,A -85,B 0,C 180,E1 30020.736,E2 30020.736} C_VEL
LIN {X 0,Y 641.646,Z 338.039,A -85,B 0,C 180,E1 30020.55,E2 30020.55} C_VEL
LIN {X 0,Y 645.038,Z 342.328,A -85,B 0,C 180,E1 30020.108,E2 30020.108} C_VEL
LIN {X 0,Y 649.19,Z 347.738,A -85,B 0,C 180,E1 30019.576,E2 30019.576} C_VEL
LIN {X 0,Y 662.488,Z 366.144,A -85,B 0,C 180,E1 30017.937,E2 30017.937} C_VEL
LIN {X 0,Y 666.933,Z 373.264,A -85,B 0,C 180,E1 30017.4,E2 30017.4} C_VEL
LIN {X 0,Y 666.647,Z 388.952,A -85,B 0,C 180,E1 30017.182,E2 30017.182} C_VEL
LIN {X 0,Y 665.835,Z 396.655,A -85,B 0,C 180,E1 30017.138,E2 30017.138} C_VEL
LIN {X 0,Y 661.154,Z 417.341,A -85,B 0,C 180,E1 30017.254,E2 30017.254} C_VEL
LIN {X 0,Y 660.488,Z 423.954,A -85,B 0,C 180,E1 30017.213,E2 30017.213} C_VEL
LIN {X 0,Y 656.24,Z 637.35,A -85,B 0,C 180,E1 30014.317,E2 30014.317} C_VEL
LIN {X 0,Y 653.107,Z 797.725,A -85,B 0,C 180,E1 30012.175,E2 30012.175} C_VEL
LIN {X 0,Y 652.021,Z 824.481,A -85,B 0,C 180,E1 30011.69,E2 30011.69} C_VEL
LIN {X 0,Y 650.474,Z 851.031,A -85,B 0,C 180,E1 30011.029,E2 30011.029} C_VEL
LIN {X 0,Y 648.981,Z 872.983,A -85,B 0,C 180,E1 30010.35,E2 30010.35} C_VEL
LIN {X 0,Y 647.39,Z 893.977,A -85,B 0,C 180,E1 30009.583,E2 30009.583} C_VEL
LIN {X 0,Y 645.425,Z 917.602,A -85,B 0,C 180,E1 30008.574,E2 30008.574} C_VEL
LIN {X 0,Y 643.116,Z 942.429,A -85,B 0,C 180,E1 30007.325,E2 30007.325} C_VEL
LIN {X 0,Y 641.046,Z 963.161,A -85,B 0,C 180,E1 30006.127,E2 30006.127} C_VEL
LIN {X 0,Y 639.157,Z 981.66,A -85,B 0,C 180,E1 30004.928,E2 30004.928} C_VEL
LIN {X 0,Y 637.132,Z 1001.013,A -85,B 0,C 180,E1 30003.532,E2 30003.532} C_VEL
LIN {X 0,Y 634.69,Z 1024.146,A -85,B 0,C 180,E1 30001.641,E2 30001.641} C_VEL
LIN {X 0,Y 632.885,Z 1041.604,A -85,B 0,C 180,E1 30000.027,E2 30000.027} C_VEL
LIN {X 0,Y 631.264,Z 1057.832,A -85,B 0,C 180,E1 29998.37,E2 29998.37} C_VEL
LIN {X 0,Y 629.509,Z 1076.059,A -85,B 0,C 180,E1 29996.304,E2 29996.304} C_VEL
LIN {X 0,Y 628.036,Z 1092.673,A -85,B 0,C 180,E1 29994.152,E2 29994.152} C_VEL
LIN {X 0,Y 626.951,Z 1106.092,A -85,B 0,C 180,E1 29992.208,E2 29992.208} C_VEL
LIN {X 0,Y 625.952,Z 1120.333,A -85,B 0,C 180,E1 29989.891,E2 29989.891} C_VEL
LIN {X 0,Y 625.169,Z 1132.935,A -85,B 0,C 180,E1 29987.498,E2 29987.498} C_VEL
LIN {X 0,Y 624.689,Z 1142.118,A -85,B 0,C 180,E1 29985.503,E2 29985.503} C_VEL
LIN {X 0,Y 624.376,Z 1150.053,A -85,B 0,C 180,E1 29983.521,E2 29983.521} C_VEL
LIN {X 0,Y 624.137,Z 1157.75,A -85,B 0,C 180,E1 29981.271,E2 29981.271} C_VEL
LIN {X 0,Y 624.001,Z 1164.589,A -85,B 0,C 180,E1 29978.756,E2 29978.756} C_VEL
LIN {X 0,Y 623.941,Z 1169.32,A -85,B 0,C 180,E1 29976.441,E2 29976.441} C_VEL
LIN {X 0,Y 623.919,Z 1172.637,A -85,B 0,C 180,E1 29974.135,E2 29974.135} C_VEL
LIN {X 0,Y 623.907,Z 1174.59,A -85,B 0,C 180,E1 29971.653,E2 29971.653} C_VEL
LIN {X 0,Y 623.894,Z 1174.86,A -85,B 0,C 180,E1 29969.357,E2 29969.357} C_VEL
LIN {X 0,Y 623.909,Z 1173.969,A -85,B 0,C 180,E1 29967.244,E2 29967.244} C_VEL
LIN {X 0,Y 623.922,Z 1171.614,A -85,B 0,C 180,E1 29964.943,E2 29964.943} C_VEL
LIN {X 0,Y 623.953,Z 1167.442,A -85,B 0,C 180,E1 29962.449,E2 29962.449} C_VEL
LIN {X 0,Y 624.05,Z 1161.741,A -85,B 0,C 180,E1 29960.036,E2 29960.036} C_VEL
LIN {X 0,Y 624.221,Z 1154.731,A -85,B 0,C 180,E1 29957.7,E2 29957.7} C_VEL
LIN {X 0,Y 624.595,Z 1144.932,A -85,B 0,C 180,E1 29955.065,E2 29955.065} C_VEL
LIN {X 0,Y 625.069,Z 1134.752,A -85,B 0,C 180,E1 29952.787,E2 29952.787} C_VEL
LIN {X 0,Y 625.672,Z 1124.481,A -85,B 0,C 180,E1 29950.78,E2 29950.78} C_VEL
LIN {X 0,Y 626.536,Z 1111.634,A -85,B 0,C 180,E1 29948.565,E2 29948.565} C_VEL
LIN {X 0,Y 627.733,Z 1096.112,A -85,B 0,C 180,E1 29946.235,E2 29946.235} C_VEL
LIN {X 0,Y 629.026,Z 1081.427,A -85,B 0,C 180,E1 29944.282,E2 29944.282} C_VEL
LIN {X 0,Y 630.635,Z 1064.105,A -85,B 0,C 180,E1 29942.217,E2 29942.217} C_VEL
LIN {X 0,Y 632.564,Z 1044.891,A -85,B 0,C 180,E1 29940.205,E2 29940.205} C_VEL
LIN {X 0,Y 634.244,Z 1028.42,A -85,B 0,C 180,E1 29938.652,E2 29938.652} C_VEL
LIN {X 0,Y 636.088,Z 1010.92,A -85,B 0,C 180,E1 29937.16,E2 29937.16} C_VEL
LIN {X 0,Y 638.427,Z 988.714,A -85,B 0,C 180,E1 29935.463,E2 29935.463} C_VEL
LIN {X 0,Y 640.745,Z 966.11,A -85,B 0,C 180,E1 29933.964,E2 29933.964} C_VEL
LIN {X 0,Y 642.713,Z 946.337,A -85,B 0,C 180,E1 29932.801,E2 29932.801} C_VEL
LIN {X 0,Y 644.731,Z 925.126,A -85,B 0,C 180,E1 29931.697,E2 29931.697} C_VEL
LIN {X 0,Y 646.96,Z 899.999,A -85,B 0,C 180,E1 29930.566,E2 29930.566} C_VEL
LIN {X 0,Y 648.76,Z 876.022,A -85,B 0,C 180,E1 29929.662,E2 29929.662} C_VEL
LIN {X 0,Y 650.289,Z 853.8,A -85,B 0,C 180,E1 29928.96,E2 29928.96} C_VEL
LIN {X 0,Y 651.63,Z 831.087,A -85,B 0,C 180,E1 29928.372,E2 29928.372} C_VEL
LIN {X 0,Y 652.943,Z 803.632,A -85,B 0,C 180,E1 29927.825,E2 29927.825} C_VEL
LIN {X 0,Y 654.039,Z 756.281,A -85,B 0,C 180,E1 29927.173,E2 29927.173} C_VEL
LIN {X 0,Y 658.276,Z 532.465,A -85,B 0,C 180,E1 29924.182,E2 29924.182} C_VEL
LIN {X 0,Y 661.378,Z 376.655,A -85,B 0,C 180,E1 29922.033,E2 29922.033} C_VEL
LIN {X 0,Y 654.601,Z 366.683,A -85,B 0,C 180,E1 29921.203,E2 29921.203} C_VEL
LIN {X 0,Y 644.533,Z 353.078,A -85,B 0,C 180,E1 29919.931,E2 29919.931} C_VEL
LIN {X 0,Y 636.66,Z 342.755,A -85,B 0,C 180,E1 29918.89,E2 29918.89} C_VEL
LIN {X 0,Y 632.791,Z 337.739,A -85,B 0,C 180,E1 29918.36,E2 29918.36} C_VEL
LIN {X 0,Y 629.899,Z 334.243,A -85,B 0,C 180,E1 29917.96,E2 29917.96} C_VEL
LIN {X 0,Y 628.862,Z 332.339,A -85,B 0,C 180,E1 29917.803,E2 29917.803} C_VEL
LIN {X 0,Y 626.218,Z 329.842,A -85,B 0,C 180,E1 29917.442,E2 29917.442} C_VEL
LIN {X 0,Y 624.957,Z 326.768,A -85,B 0,C 180,E1 29917.232,E2 29917.232} C_VEL
LIN {X 0,Y 624.898,Z 326.387,A -85,B 0,C 180,E1 29917.217,E2 29917.217} C_VEL
LIN {X 0,Y 624.845,Z 326.364,A -85,B 0,C 180,E1 29914.342,E2 29914.342} C_VEL
LIN {X 0,Y 624.928,Z 326.364,A -85,B 0,C 180,E1 29911.309,E2 29911.309} C_VEL
LIN {X 0,Y 624.853,Z 326.394,A -85,B 0,C 180,E1 29908.348,E2 29908.348} C_VEL
LIN {X 0,Y 624.921,Z 326.355,A -85,B 0,C 180,E1 29905.392,E2 29905.392} C_VEL
LIN {X 0,Y 624.861,Z 326.391,A -85,B 0,C 180,E1 29902.351,E2 29902.351} C_VEL
LIN {X 0,Y 624.88,Z 326.359,A -85,B 0,C 180,E1 29899.635,E2 29899.635} C_VEL
LIN {X 0,Y 624.88,Z 326.381,A -85,B 0,C 180,E1 29896.453,E2 29896.453} C_VEL
LIN {X 0,Y 624.87,Z 326.368,A -85,B 0,C 180,E1 29893.77,E2 29893.77} C_VEL
LIN {X 0,Y 624.93,Z 326.374,A -85,B 0,C 180,E1 29890.696,E2 29890.696} C_VEL
LIN {X 0,Y 624.873,Z 326.369,A -85,B 0,C 180,E1 29887.817,E2 29887.817} C_VEL
LIN {X 0,Y 624.949,Z 326.376,A -85,B 0,C 180,E1 29884.864,E2 29884.864} C_VEL
LIN {X 0,Y 624.88,Z 326.365,A -85,B 0,C 180,E1 29881.834,E2 29881.834} C_VEL
LIN {X 0,Y 624.927,Z 326.384,A -85,B 0,C 180,E1 29878.992,E2 29878.992} C_VEL
LIN {X 0,Y 624.893,Z 326.361,A -85,B 0,C 180,E1 29875.871,E2 29875.871} C_VEL
LIN {X 0,Y 624.914,Z 326.387,A -85,B 0,C 180,E1 29873.015,E2 29873.015} C_VEL
LIN {X 0,Y 624.9,Z 326.365,A -85,B 0,C 180,E1 29869.742,E2 29869.742} C_VEL
LIN {X 0,Y 624.92,Z 326.378,A -85,B 0,C 180,E1 29866.867,E2 29866.867} C_VEL
LIN {X 0,Y 624.91,Z 326.376,A -85,B 0,C 180,E1 29863.644,E2 29863.644} C_VEL
LIN {X 0,Y 624.93,Z 326.36,A -85,B 0,C 180,E1 29860.658,E2 29860.658} C_VEL
LIN {X 0,Y 624.911,Z 326.387,A -85,B 0,C 180,E1 29857.417,E2 29857.417} C_VEL
LIN {X 0,Y 624.944,Z 326.354,A -85,B 0,C 180,E1 29854.406,E2 29854.406} C_VEL
LIN {X 0,Y 624.915,Z 326.37,A -85,B 0,C 180,E1 29851.258,E2 29851.258} C_VEL
LIN {X 0,Y 624.952,Z 326.387,A -85,B 0,C 180,E1 29848.238,E2 29848.238} C_VEL
LIN {X 0,Y 624.918,Z 326.37,A -85,B 0,C 180,E1 29845.053,E2 29845.053} C_VEL
LIN {X 0,Y 624.953,Z 326.634,A -85,B 0,C 180,E1 29844.831,E2 29844.831} C_VEL
LIN {X 0,Y 626.257,Z 329.888,A -85,B 0,C 180,E1 29844.355,E2 29844.355} C_VEL
LIN {X 0,Y 627.365,Z 331.57,A -85,B 0,C 180,E1 29844.059,E2 29844.059} C_VEL
LIN {X 0,Y 634.279,Z 345.706,A -85,B 0,C 180,E1 29841.947,E2 29841.947} C_VEL
LIN {X 0,Y 636.116,Z 349.178,A -85,B 0,C 180,E1 29841.475,E2 29841.475} C_VEL
LIN {X 0,Y 650.959,Z 370.445,A -85,B 0,C 180,E1 29839.521,E2 29839.521} C_VEL
LIN {X 0,Y 661.485,Z 386.133,A -85,B 0,C 180,E1 29838.223,E2 29838.223} C_VEL
LIN {X 0,Y 661.775,Z 388.907,A -85,B 0,C 180,E1 29838.151,E2 29838.151} C_VEL
LIN {X 0,Y 657.625,Z 595.41,A -85,B 0,C 180,E1 29835.328,E2 29835.328} C_VEL
LIN {X 0,Y 653.42,Z 818.257,A -85,B 0,C 180,E1 29832.359,E2 29832.359} C_VEL
LIN {X 0,Y 652.483,Z 843.447,A -85,B 0,C 180,E1 29831.952,E2 29831.952} C_VEL
LIN {X 0,Y 651.364,Z 865.883,A -85,B 0,C 180,E1 29831.469,E2 29831.469} C_VEL
LIN {X 0,Y 649.943,Z 889.524,A -85,B 0,C 180,E1 29830.829,E2 29830.829} C_VEL
LIN {X 0,Y 647.907,Z 917.457,A -85,B 0,C 180,E1 29829.882,E2 29829.882} C_VEL
LIN {X 0,Y 646.075,Z 939.473,A -85,B 0,C 180,E1 29828.983,E2 29828.983} C_VEL
LIN {X 0,Y 644.275,Z 959.708,A -85,B 0,C 180,E1 29828.032,E2 29828.032} C_VEL
LIN {X 0,Y 642.213,Z 981.338,A -85,B 0,C 180,E1 29826.877,E2 29826.877} C_VEL
LIN {X 0,Y 639.689,Z 1006.564,A -85,B 0,C 180,E1 29825.32,E2 29825.32} C_VEL
LIN {X 0,Y 637.634,Z 1026.241,A -85,B 0,C 180,E1 29823.934,E2 29823.934} C_VEL
LIN {X 0,Y 635.761,Z 1044.058,A -85,B 0,C 180,E1 29822.538,E2 29822.538} C_VEL
LIN {X 0,Y 633.858,Z 1062.383,A -85,B 0,C 180,E1 29820.946,E2 29820.946} C_VEL
LIN {X 0,Y 631.663,Z 1083.6,A -85,B 0,C 180,E1 29818.867,E2 29818.867} C_VEL
LIN {X 0,Y 630.112,Z 1099.691,A -85,B 0,C 180,E1 29817.091,E2 29817.091} C_VEL
LIN {X 0,Y 628.627,Z 1115.707,A -85,B 0,C 180,E1 29815.13,E2 29815.13} C_VEL
LIN {X 0,Y 627.226,Z 1132.542,A -85,B 0,C 180,E1 29812.791,E2 29812.791} C_VEL
LIN {X 0,Y 626.274,Z 1145.438,A -85,B 0,C 180,E1 29810.758,E2 29810.758} C_VEL
LIN {X 0,Y 625.493,Z 1157.337,A -85,B 0,C 180,E1 29808.645,E2 29808.645} C_VEL
LIN {X 0,Y 624.818,Z 1169.849,A -85,B 0,C 180,E1 29806.072,E2 29806.072} C_VEL
LIN {X 0,Y 624.427,Z 1178.803,A -85,B 0,C 180,E1 29803.897,E2 29803.897} C_VEL
LIN {X 0,Y 624.182,Z 1186.124,A -85,B 0,C 180,E1 29801.825,E2 29801.825} C_VEL
LIN {X 0,Y 624.028,Z 1193.109,A -85,B 0,C 180,E1 29799.406,E2 29799.406} C_VEL
LIN {X 0,Y 623.941,Z 1198.594,A -85,B 0,C 180,E1 29796.903,E2 29796.903} C_VEL
LIN {X 0,Y 623.913,Z 1202.127,A -85,B 0,C 180,E1 29794.596,E2 29794.596} C_VEL
LIN {X 0,Y 623.911,Z 1204.27,A -85,B 0,C 180,E1 29792.296,E2 29792.296} C_VEL
LIN {X 0,Y 623.897,Z 1204.939,A -85,B 0,C 180,E1 29789.725,E2 29789.725} C_VEL
LIN {X 0,Y 623.908,Z 1204.072,A -85,B 0,C 180,E1 29787.428,E2 29787.428} C_VEL
LIN {X 0,Y 623.916,Z 1201.899,A -85,B 0,C 180,E1 29785.22,E2 29785.22} C_VEL
LIN {X 0,Y 623.958,Z 1198.079,A -85,B 0,C 180,E1 29782.82,E2 29782.82} C_VEL
LIN {X 0,Y 624.038,Z 1192.377,A -85,B 0,C 180,E1 29780.315,E2 29780.315} C_VEL
LIN {X 0,Y 624.194,Z 1185.494,A -85,B 0,C 180,E1 29777.981,E2 29777.981} C_VEL
LIN {X 0,Y 624.485,Z 1177.372,A -85,B 0,C 180,E1 29775.726,E2 29775.726} C_VEL
LIN {X 0,Y 624.975,Z 1166.374,A -85,B 0,C 180,E1 29773.168,E2 29773.168} C_VEL
LIN {X 0,Y 625.586,Z 1155.797,A -85,B 0,C 180,E1 29771.068,E2 29771.068} C_VEL
LIN {X 0,Y 626.355,Z 1144.275,A -85,B 0,C 180,E1 29769.048,E2 29769.048} C_VEL
LIN {X 0,Y 627.501,Z 1129.299,A -85,B 0,C 180,E1 29766.724,E2 29766.724} C_VEL
LIN {X 0,Y 628.84,Z 1113.388,A -85,B 0,C 180,E1 29764.576,E2 29764.576} C_VEL
LIN {X 0,Y 630.262,Z 1097.999,A -85,B 0,C 180,E1 29762.711,E2 29762.711} C_VEL
LIN {X 0,Y 632.18,Z 1078.815,A -85,B 0,C 180,E1 29760.633,E2 29760.633} C_VEL
LIN {X 0,Y 634.137,Z 1059.613,A -85,B 0,C 180,E1 29758.805,E2 29758.805} C_VEL
LIN {X 0,Y 635.948,Z 1042.23,A -85,B 0,C 180,E1 29757.312,E2 29757.312} C_VEL
LIN {X 0,Y 637.971,Z 1022.963,A -85,B 0,C 180,E1 29755.821,E2 29755.821} C_VEL
LIN {X 0,Y 640.479,Z 998.678,A -85,B 0,C 180,E1 29754.168,E2 29754.168} C_VEL
LIN {X 0,Y 642.579,Z 977.651,A -85,B 0,C 180,E1 29752.918,E2 29752.918} C_VEL
LIN {X 0,Y 644.473,Z 957.703,A -85,B 0,C 180,E1 29751.868,E2 29751.868} C_VEL
LIN {X 0,Y 646.513,Z 934.954,A -85,B 0,C 180,E1 29750.82,E2 29750.82} C_VEL
LIN {X 0,Y 648.635,Z 907.83,A -85,B 0,C 180,E1 29749.768,E2 29749.768} C_VEL
LIN {X 0,Y 650.216,Z 884.874,A -85,B 0,C 180,E1 29749.035,E2 29749.035} C_VEL
LIN {X 0,Y 651.533,Z 862.754,A -85,B 0,C 180,E1 29748.456,E2 29748.456} C_VEL
LIN {X 0,Y 652.799,Z 836.952,A -85,B 0,C 180,E1 29747.926,E2 29747.926} C_VEL
LIN {X 0,Y 653.806,Z 799.115,A -85,B 0,C 180,E1 29747.387,E2 29747.387} C_VEL
LIN {X 0,Y 658.073,Z 573.016,A -85,B 0,C 180,E1 29744.37,E2 29744.37} C_VEL
LIN {X 0,Y 661.747,Z 387.252,A -85,B 0,C 180,E1 29741.82,E2 29741.82} C_VEL
LIN {X 0,Y 660.991,Z 385.134,A -85,B 0,C 180,E1 29741.714,E2 29741.714} C_VEL
LIN {X 0,Y 644.485,Z 361.065,A -85,B 0,C 180,E1 29739.646,E2 29739.646} C_VEL
LIN {X 0,Y 635.584,Z 348.192,A -85,B 0,C 180,E1 29738.419,E2 29738.419} C_VEL
LIN {X 0,Y 630.837,Z 338.827,A -85,B 0,C 180,E1 29737.036,E2 29737.036} C_VEL
LIN {X 0,Y 628.703,Z 334.546,A -85,B 0,C 180,E1 29736.386,E2 29736.386} C_VEL
LIN {X 0,Y 626.605,Z 330.353,A -85,B 0,C 180,E1 29735.735,E2 29735.735} C_VEL
LIN {X 0,Y 625.121,Z 327.424,A -85,B 0,C 180,E1 29735.27,E2 29735.27} C_VEL
LIN {X 0,Y 624.917,Z 326.374,A -85,B 0,C 180,E1 29735.095,E2 29735.095} C_VEL
LIN {X 0,Y 624.952,Z 326.384,A -85,B 0,C 180,E1 29731.977,E2 29731.977} C_VEL
LIN {X 0,Y 624.911,Z 326.365,A -85,B 0,C 180,E1 29728.932,E2 29728.932} C_VEL
LIN {X 0,Y 624.95,Z 326.356,A -85,B 0,C 180,E1 29725.899,E2 29725.899} C_VEL
LIN {X 0,Y 624.908,Z 326.389,A -85,B 0,C 180,E1 29722.839,E2 29722.839} C_VEL
LIN {X 0,Y 624.952,Z 326.35,A -85,B 0,C 180,E1 29719.73,E2 29719.73} C_VEL
LIN {X 0,Y 624.901,Z 326.382,A -85,B 0,C 180,E1 29716.643,E2 29716.643} C_VEL
LIN {X 0,Y 624.955,Z 326.36,A -85,B 0,C 180,E1 29713.603,E2 29713.603} C_VEL
LIN {X 0,Y 624.895,Z 326.375,A -85,B 0,C 180,E1 29710.604,E2 29710.604} C_VEL
LIN {X 0,Y 624.956,Z 326.365,A -85,B 0,C 180,E1 29707.539,E2 29707.539} C_VEL
LIN {X 0,Y 624.889,Z 326.373,A -85,B 0,C 180,E1 29704.497,E2 29704.497} C_VEL
LIN {X 0,Y 624.951,Z 326.367,A -85,B 0,C 180,E1 29701.467,E2 29701.467} C_VEL
LIN {X 0,Y 624.886,Z 326.373,A -85,B 0,C 180,E1 29698.441,E2 29698.441} C_VEL
LIN {X 0,Y 624.929,Z 326.368,A -85,B 0,C 180,E1 29695.503,E2 29695.503} C_VEL
LIN {X 0,Y 624.886,Z 326.373,A -85,B 0,C 180,E1 29692.368,E2 29692.368} C_VEL
LIN {X 0,Y 624.898,Z 326.371,A -85,B 0,C 180,E1 29689.583,E2 29689.583} C_VEL
LIN {X 0,Y 624.888,Z 326.371,A -85,B 0,C 180,E1 29686.396,E2 29686.396} C_VEL
LIN {X 0,Y 624.874,Z 326.378,A -85,B 0,C 180,E1 29683.738,E2 29683.738} C_VEL
LIN {X 0,Y 624.927,Z 326.362,A -85,B 0,C 180,E1 29680.658,E2 29680.658} C_VEL
LIN {X 0,Y 624.865,Z 326.389,A -85,B 0,C 180,E1 29677.812,E2 29677.812} C_VEL
LIN {X 0,Y 624.922,Z 326.359,A -85,B 0,C 180,E1 29674.912,E2 29674.912} C_VEL
LIN {X 0,Y 624.864,Z 326.394,A -85,B 0,C 180,E1 29671.832,E2 29671.832} C_VEL
LIN {X 0,Y 624.868,Z 326.361,A -85,B 0,C 180,E1 29669.199,E2 29669.199} C_VEL
LIN {X 0,Y 624.868,Z 326.365,A -85,B 0,C 180,E1 29665.94,E2 29665.94} C_VEL
LIN {X 0,Y 624.856,Z 326.399,A -85,B 0,C 180,E1 29663.239,E2 29663.239} C_VEL
LIN {X 0,Y 624.92,Z 326.496,A -85,B 0,C 180,E1 29662.686,E2 29662.686} C_VEL
LIN {X 0,Y 626.064,Z 329.589,A -85,B 0,C 180,E1 29662.49,E2 29662.49} C_VEL
LIN {X 0,Y 628.695,Z 332.223,A -85,B 0,C 180,E1 29662.128,E2 29662.128} C_VEL
LIN {X 0,Y 631.922,Z 336.917,A -85,B 0,C 180,E1 29661.665,E2 29661.665} C_VEL
LIN {X 0,Y 633.813,Z 338.96,A -85,B 0,C 180,E1 29661.41,E2 29661.41} C_VEL
LIN {X 0,Y 637.217,Z 343.278,A -85,B 0,C 180,E1 29660.949,E2 29660.949} C_VEL
LIN {X 0,Y 641.418,Z 348.799,A -85,B 0,C 180,E1 29660.388,E2 29660.388} C_VEL
LIN {X 0,Y 656.929,Z 369.818,A -85,B 0,C 180,E1 29658.423,E2 29658.423} C_VEL
LIN {X 0,Y 661.467,Z 377.123,A -85,B 0,C 180,E1 29657.861,E2 29657.861} C_VEL
LIN {X 0,Y 660.488,Z 423.954,A -85,B 0,C 180,E1 29657.213,E2 29657.213} C_VEL
LIN {X 0,Y 659.631,Z 431.662,A -85,B 0,C 180,E1 29657.172,E2 29657.172} C_VEL
LIN {X 0,Y 654.95,Z 452.344,A -85,B 0,C 180,E1 29657.29,E2 29657.29} C_VEL
LIN {X 0,Y 654.312,Z 458.951,A -85,B 0,C 180,E1 29657.246,E2 29657.246} C_VEL
LIN {X 0,Y 649.76,Z 674.985,A -85,B 0,C 180,E1 29654.306,E2 29654.306} C_VEL
LIN {X 0,Y 647.171,Z 797.952,A -85,B 0,C 180,E1 29652.649,E2 29652.649} C_VEL
LIN {X 0,Y 645.999,Z 825.033,A -85,B 0,C 180,E1 29652.154,E2 29652.154} C_VEL
LIN {X 0,Y 644.366,Z 851.373,A -85,B 0,C 180,E1 29651.492,E2 29651.492} C_VEL
LIN {X 0,Y 642.809,Z 872.999,A -85,B 0,C 180,E1 29650.819,E2 29650.819} C_VEL
LIN {X 0,Y 641.194,Z 892.888,A -85,B 0,C 180,E1 29650.092,E2 29650.092} C_VEL
LIN {X 0,Y 639.198,Z 915.378,A -85,B 0,C 180,E1 29649.136,E2 29649.136} C_VEL
LIN {X 0,Y 636.641,Z 941.746,A -85,B 0,C 180,E1 29647.814,E2 29647.814} C_VEL
LIN {X 0,Y 634.456,Z 962.357,A -85,B 0,C 180,E1 29646.619,E2 29646.619} C_VEL
LIN {X 0,Y 632.427,Z 980.932,A -85,B 0,C 180,E1 29645.41,E2 29645.41} C_VEL
LIN {X 0,Y 630.339,Z 999.691,A -85,B 0,C 180,E1 29644.051,E2 29644.051} C_VEL
LIN {X 0,Y 627.869,Z 1021.727,A -85,B 0,C 180,E1 29642.26,E2 29642.26} C_VEL
LIN {X 0,Y 625.644,Z 1041.358,A -85,B 0,C 180,E1 29640.438,E2 29640.438} C_VEL
LIN {X 0,Y 623.874,Z 1057.837,A -85,B 0,C 180,E1 29638.737,E2 29638.737} C_VEL
LIN {X 0,Y 622.001,Z 1076.073,A -85,B 0,C 180,E1 29636.646,E2 29636.646} C_VEL
LIN {X 0,Y 620.361,Z 1093.146,A -85,B 0,C 180,E1 29634.403,E2 29634.403} C_VEL
LIN {X 0,Y 619.171,Z 1106.729,A -85,B 0,C 180,E1 29632.402,E2 29632.402} C_VEL
LIN {X 0,Y 618.057,Z 1121.399,A -85,B 0,C 180,E1 29629.958,E2 29629.958} C_VEL
LIN {X 0,Y 617.281,Z 1132.94,A -85,B 0,C 180,E1 29627.729,E2 29627.729} C_VEL
LIN {X 0,Y 616.746,Z 1142.525,A -85,B 0,C 180,E1 29625.612,E2 29625.612} C_VEL
LIN {X 0,Y 616.396,Z 1150.761,A -85,B 0,C 180,E1 29623.508,E2 29623.508} C_VEL
LIN {X 0,Y 616.132,Z 1158.627,A -85,B 0,C 180,E1 29621.134,E2 29621.134} C_VEL
LIN {X 0,Y 616.002,Z 1165.219,A -85,B 0,C 180,E1 29618.588,E2 29618.588} C_VEL
LIN {X 0,Y 615.943,Z 1169.637,A -85,B 0,C 180,E1 29616.337,E2 29616.337} C_VEL
LIN {X 0,Y 615.915,Z 1172.943,A -85,B 0,C 180,E1 29613.91,E2 29613.91} C_VEL
LIN {X 0,Y 615.908,Z 1174.635,A -85,B 0,C 180,E1 29611.488,E2 29611.488} C_VEL
LIN {X 0,Y 615.894,Z 1174.86,A -85,B 0,C 180,E1 29609.349,E2 29609.349} C_VEL
LIN {X 0,Y 615.91,Z 1173.966,A -85,B 0,C 180,E1 29607.209,E2 29607.209} C_VEL
LIN {X 0,Y 615.922,Z 1171.61,A -85,B 0,C 180,E1 29604.878,E2 29604.878} C_VEL
LIN {X 0,Y 615.96,Z 1167.441,A -85,B 0,C 180,E1 29602.351,E2 29602.351} C_VEL
LIN {X 0,Y 616.066,Z 1161.736,A -85,B 0,C 180,E1 29599.905,E2 29599.905} C_VEL
LIN {X 0,Y 616.243,Z 1155.02,A -85,B 0,C 180,E1 29597.63,E2 29597.63} C_VEL
LIN {X 0,Y 616.629,Z 1145.738,A -85,B 0,C 180,E1 29595.059,E2 29595.059} C_VEL
LIN {X 0,Y 617.17,Z 1134.952,A -85,B 0,C 180,E1 29592.603,E2 29592.603} C_VEL
LIN {X 0,Y 617.839,Z 1124.479,A -85,B 0,C 180,E1 29590.526,E2 29590.526} C_VEL
LIN {X 0,Y 618.833,Z 1111.05,A -85,B 0,C 180,E1 29588.185,E2 29588.185} C_VEL
LIN {X 0,Y 620.143,Z 1095.405,A -85,B 0,C 180,E1 29585.825,E2 29585.825} C_VEL
LIN {X 0,Y 621.529,Z 1080.649,A -85,B 0,C 180,E1 29583.846,E2 29583.846} C_VEL
LIN {X 0,Y 623.463,Z 1061.995,A -85,B 0,C 180,E1 29581.622,E2 29581.622} C_VEL
LIN {X 0,Y 625.406,Z 1043.605,A -85,B 0,C 180,E1 29579.695,E2 29579.695} C_VEL
LIN {X 0,Y 627.268,Z 1026.747,A -85,B 0,C 180,E1 29578.102,E2 29578.102} C_VEL
LIN {X 0,Y 629.68,Z 1005.67,A -85,B 0,C 180,E1 29576.313,E2 29576.313} C_VEL
LIN {X 0,Y 632.135,Z 983.673,A -85,B 0,C 180,E1 29574.687,E2 29574.687} C_VEL
LIN {X 0,Y 634.229,Z 964.473,A -85,B 0,C 180,E1 29573.422,E2 29573.422} C_VEL
LIN {X 0,Y 636.223,Z 945.66,A -85,B 0,C 180,E1 29572.314,E2 29572.314} C_VEL
LIN {X 0,Y 638.366,Z 924.461,A -85,B 0,C 180,E1 29571.207,E2 29571.207} C_VEL
LIN {X 0,Y 640.758,Z 898.713,A -85,B 0,C 180,E1 29570.05,E2 29570.05} C_VEL
LIN {X 0,Y 642.58,Z 876,A -85,B 0,C 180,E1 29569.192,E2 29569.192} C_VEL
LIN {X 0,Y 644.184,Z 854,A -85,B 0,C 180,E1 29568.494,E2 29568.494} C_VEL
LIN {X 0,Y 645.57,Z 831.823,A -85,B 0,C 180,E1 29567.914,E2 29567.914} C_VEL
LIN {X 0,Y 646.951,Z 805.124,A -85,B 0,C 180,E1 29567.372,E2 29567.372} C_VEL
LIN {X 0,Y 648.057,Z 761.958,A -85,B 0,C 180,E1 29566.766,E2 29566.766} C_VEL
LIN {X 0,Y 652.596,Z 538.065,A -85,B 0,C 180,E1 29563.752,E2 29563.752} C_VEL
LIN {X 0,Y 655.969,Z 380.426,A -85,B 0,C 180,E1 29561.564,E2 29561.564} C_VEL
LIN {X 0,Y 648.165,Z 369.273,A -85,B 0,C 180,E1 29560.588,E2 29560.588} C_VEL
LIN {X 0,Y 640.049,Z 358.423,A -85,B 0,C 180,E1 29559.539,E2 29559.539} C_VEL
LIN {X 0,Y 632.803,Z 348.883,A -85,B 0,C 180,E1 29558.561,E2 29558.561} C_VEL
LIN {X 0,Y 629.098,Z 344.114,A -85,B 0,C 180,E1 29558.046,E2 29558.046} C_VEL
LIN {X 0,Y 625.857,Z 339.777,A -85,B 0,C 180,E1 29557.582,E2 29557.582} C_VEL
LIN {X 0,Y 622.08,Z 335.204,A -85,B 0,C 180,E1 29557.038,E2 29557.038} C_VEL
LIN {X 0,Y 621.2,Z 333.505,A -85,B 0,C 180,E1 29556.898,E2 29556.898} C_VEL
LIN {X 0,Y 618.453,Z 331.201,A -85,B 0,C 180,E1 29556.511,E2 29556.511} C_VEL
LIN {X 0,Y 617.04,Z 328.11,A -85,B 0,C 180,E1 29556.272,E2 29556.272} C_VEL
LIN {X 0,Y 616.917,Z 327.382,A -85,B 0,C 180,E1 29556.238,E2 29556.238} C_VEL
LIN {X 0,Y 616.949,Z 327.37,A -85,B 0,C 180,E1 29553.084,E2 29553.084} C_VEL
LIN {X 0,Y 616.907,Z 327.349,A -85,B 0,C 180,E1 29550.247,E2 29550.247} C_VEL
LIN {X 0,Y 616.995,Z 327.368,A -85,B 0,C 180,E1 29547.299,E2 29547.299} C_VEL
LIN {X 0,Y 616.918,Z 327.367,A -85,B 0,C 180,E1 29544.311,E2 29544.311} C_VEL
LIN {X 0,Y 616.955,Z 327.355,A -85,B 0,C 180,E1 29541.528,E2 29541.528} C_VEL
LIN {X 0,Y 616.931,Z 327.379,A -85,B 0,C 180,E1 29538.326,E2 29538.326} C_VEL
LIN {X 0,Y 616.941,Z 327.351,A -85,B 0,C 180,E1 29535.607,E2 29535.607} C_VEL
LIN {X 0,Y 616.947,Z 327.379,A -85,B 0,C 180,E1 29532.353,E2 29532.353} C_VEL
LIN {X 0,Y 616.937,Z 327.349,A -85,B 0,C 180,E1 29529.61,E2 29529.61} C_VEL
LIN {X 0,Y 616.974,Z 327.377,A -85,B 0,C 180,E1 29526.42,E2 29526.42} C_VEL
LIN {X 0,Y 616.941,Z 327.348,A -85,B 0,C 180,E1 29523.531,E2 29523.531} C_VEL
LIN {X 0,Y 616.992,Z 327.376,A -85,B 0,C 180,E1 29520.371,E2 29520.371} C_VEL
LIN {X 0,Y 616.947,Z 327.35,A -85,B 0,C 180,E1 29517.492,E2 29517.492} C_VEL
LIN {X 0,Y 617.007,Z 327.372,A -85,B 0,C 180,E1 29514.327,E2 29514.327} C_VEL
LIN {X 0,Y 616.951,Z 327.347,A -85,B 0,C 180,E1 29511.425,E2 29511.425} C_VEL
LIN {X 0,Y 617.016,Z 327.373,A -85,B 0,C 180,E1 29508.313,E2 29508.313} C_VEL
LIN {X 0,Y 616.956,Z 327.342,A -85,B 0,C 180,E1 29505.259,E2 29505.259} C_VEL
LIN {X 0,Y 617.017,Z 327.371,A -85,B 0,C 180,E1 29502.165,E2 29502.165} C_VEL
LIN {X 0,Y 616.963,Z 327.345,A -85,B 0,C 180,E1 29499.112,E2 29499.112} C_VEL
LIN {X 0,Y 617.014,Z 327.356,A -85,B 0,C 180,E1 29496.057,E2 29496.057} C_VEL
LIN {X 0,Y 616.97,Z 327.373,A -85,B 0,C 180,E1 29493.013,E2 29493.013} C_VEL
LIN {X 0,Y 617.011,Z 327.34,A -85,B 0,C 180,E1 29489.921,E2 29489.921} C_VEL
LIN {X 0,Y 616.973,Z 327.352,A -85,B 0,C 180,E1 29486.896,E2 29486.896} C_VEL
LIN {X 0,Y 617.033,Z 327.523,A -85,B 0,C 180,E1 29485.755,E2 29485.755} C_VEL
LIN {X 0,Y 618.466,Z 331.087,A -85,B 0,C 180,E1 29485.212,E2 29485.212} C_VEL
LIN {X 0,Y 619.49,Z 332.772,A -85,B 0,C 180,E1 29484.915,E2 29484.915} C_VEL
LIN {X 0,Y 624.487,Z 342.881,A -85,B 0,C 180,E1 29483.328,E2 29483.328} C_VEL
LIN {X 0,Y 627.501,Z 348.653,A -85,B 0,C 180,E1 29482.476,E2 29482.476} C_VEL
LIN {X 0,Y 639.51,Z 365.591,A -85,B 0,C 180,E1 29480.812,E2 29480.812} C_VEL
LIN {X 0,Y 654.683,Z 387.771,A -85,B 0,C 180,E1 29478.861,E2 29478.861} C_VEL
LIN {X 0,Y 656.373,Z 390.656,A -85,B 0,C 180,E1 29478.648,E2 29478.648} C_VEL
LIN {X 0,Y 651.959,Z 596.982,A -85,B 0,C 180,E1 29475.808,E2 29475.808} C_VEL
LIN {X 0,Y 647.485,Z 818.859,A -85,B 0,C 180,E1 29472.828,E2 29472.828} C_VEL
LIN {X 0,Y 646.517,Z 843.422,A -85,B 0,C 180,E1 29472.429,E2 29472.429} C_VEL
LIN {X 0,Y 645.344,Z 865.655,A -85,B 0,C 180,E1 29471.949,E2 29471.949} C_VEL
LIN {X 0,Y 643.868,Z 888.748,A -85,B 0,C 180,E1 29471.324,E2 29471.324} C_VEL
LIN {X 0,Y 641.709,Z 917.053,A -85,B 0,C 180,E1 29470.364,E2 29470.364} C_VEL
LIN {X 0,Y 639.767,Z 939.131,A -85,B 0,C 180,E1 29469.459,E2 29469.459} C_VEL
LIN {X 0,Y 637.819,Z 959.705,A -85,B 0,C 180,E1 29468.487,E2 29468.487} C_VEL
LIN {X 0,Y 635.633,Z 981.251,A -85,B 0,C 180,E1 29467.329,E2 29467.329} C_VEL
LIN {X 0,Y 632.925,Z 1006.392,A -85,B 0,C 180,E1 29465.768,E2 29465.768} C_VEL
LIN {X 0,Y 630.713,Z 1026.238,A -85,B 0,C 180,E1 29464.358,E2 29464.358} C_VEL
LIN {X 0,Y 628.713,Z 1044.056,A -85,B 0,C 180,E1 29462.949,E2 29462.949} C_VEL
LIN {X 0,Y 626.561,Z 1063.49,A -85,B 0,C 180,E1 29461.24,E2 29461.24} C_VEL
LIN {X 0,Y 624.267,Z 1083.986,A -85,B 0,C 180,E1 29459.199,E2 29459.199} C_VEL
LIN {X 0,Y 622.628,Z 1099.689,A -85,B 0,C 180,E1 29457.444,E2 29457.444} C_VEL
LIN {X 0,Y 621.012,Z 1116.091,A -85,B 0,C 180,E1 29455.409,E2 29455.409} C_VEL
LIN {X 0,Y 619.468,Z 1133.188,A -85,B 0,C 180,E1 29452.992,E2 29452.992} C_VEL
LIN {X 0,Y 618.444,Z 1146.009,A -85,B 0,C 180,E1 29450.934,E2 29450.934} C_VEL
LIN {X 0,Y 617.578,Z 1158.365,A -85,B 0,C 180,E1 29448.697,E2 29448.697} C_VEL
LIN {X 0,Y 616.881,Z 1170.261,A -85,B 0,C 180,E1 29446.187,E2 29446.187} C_VEL
LIN {X 0,Y 616.475,Z 1178.805,A -85,B 0,C 180,E1 29444.08,E2 29444.08} C_VEL
LIN {X 0,Y 616.204,Z 1186.098,A -85,B 0,C 180,E1 29441.987,E2 29441.987} C_VEL
LIN {X 0,Y 616.039,Z 1193.109,A -85,B 0,C 180,E1 29439.529,E2 29439.529} C_VEL
LIN {X 0,Y 615.947,Z 1198.594,A -85,B 0,C 180,E1 29436.993,E2 29436.993} C_VEL
LIN {X 0,Y 615.914,Z 1202.124,A -85,B 0,C 180,E1 29434.656,E2 29434.656} C_VEL
LIN {X 0,Y 615.911,Z 1204.27,A -85,B 0,C 180,E1 29432.326,E2 29432.326} C_VEL
LIN {X 0,Y 615.897,Z 1204.939,A -85,B 0,C 180,E1 29429.721,E2 29429.721} C_VEL
LIN {X 0,Y 615.909,Z 1204.069,A -85,B 0,C 180,E1 29427.395,E2 29427.395} C_VEL
LIN {X 0,Y 615.918,Z 1201.896,A -85,B 0,C 180,E1 29425.158,E2 29425.158} C_VEL
LIN {X 0,Y 615.961,Z 1197.989,A -85,B 0,C 180,E1 29422.677,E2 29422.677} C_VEL
LIN {X 0,Y 616.053,Z 1192.224,A -85,B 0,C 180,E1 29420.131,E2 29420.131} C_VEL
LIN {X 0,Y 616.22,Z 1185.491,A -85,B 0,C 180,E1 29417.823,E2 29417.823} C_VEL
LIN {X 0,Y 616.552,Z 1177.267,A -85,B 0,C 180,E1 29415.509,E2 29415.509} C_VEL
LIN {X 0,Y 617.081,Z 1166.36,A -85,B 0,C 180,E1 29412.943,E2 29412.943} C_VEL
LIN {X 0,Y 617.736,Z 1155.795,A -85,B 0,C 180,E1 29410.818,E2 29410.818} C_VEL
LIN {X 0,Y 618.572,Z 1144.283,A -85,B 0,C 180,E1 29408.773,E2 29408.773} C_VEL
LIN {X 0,Y 619.831,Z 1129.089,A -85,B 0,C 180,E1 29406.389,E2 29406.389} C_VEL
LIN {X 0,Y 621.28,Z 1113.393,A -85,B 0,C 180,E1 29404.245,E2 29404.245} C_VEL
LIN {X 0,Y 622.789,Z 1097.999,A -85,B 0,C 180,E1 29402.356,E2 29402.356} C_VEL
LIN {X 0,Y 624.875,Z 1078.882,A -85,B 0,C 180,E1 29400.262,E2 29400.262} C_VEL
LIN {X 0,Y 626.91,Z 1060.167,A -85,B 0,C 180,E1 29398.458,E2 29398.458} C_VEL
LIN {X 0,Y 628.843,Z 1042.837,A -85,B 0,C 180,E1 29396.95,E2 29396.95} C_VEL
LIN {X 0,Y 630.916,Z 1024.336,A -85,B 0,C 180,E1 29395.499,E2 29395.499} C_VEL
LIN {X 0,Y 633.6,Z 1000.286,A -85,B 0,C 180,E1 29393.829,E2 29393.829} C_VEL
LIN {X 0,Y 635.914,Z 978.548,A -85,B 0,C 180,E1 29392.52,E2 29392.52} C_VEL
LIN {X 0,Y 637.938,Z 958.562,A -85,B 0,C 180,E1 29391.456,E2 29391.456} C_VEL
LIN {X 0,Y 639.961,Z 937.213,A -85,B 0,C 180,E1 29390.456,E2 29390.456} C_VEL
LIN {X 0,Y 642.286,Z 910.041,A -85,B 0,C 180,E1 29389.376,E2 29389.376} C_VEL
LIN {X 0,Y 644.068,Z 885.644,A -85,B 0,C 180,E1 29388.586,E2 29388.586} C_VEL
LIN {X 0,Y 645.451,Z 863.788,A -85,B 0,C 180,E1 29388.006,E2 29388.006} C_VEL
LIN {X 0,Y 646.658,Z 840.519,A -85,B 0,C 180,E1 29387.516,E2 29387.516} C_VEL
LIN {X 0,Y 647.768,Z 806.802,A -85,B 0,C 180,E1 29387.008,E2 29387.008} C_VEL
LIN {X 0,Y 652.248,Z 583.143,A -85,B 0,C 180,E1 29384.004,E2 29384.004} C_VEL
LIN {X 0,Y 656.354,Z 390.295,A -85,B 0,C 180,E1 29381.345,E2 29381.345} C_VEL
LIN {X 0,Y 640.561,Z 367.073,A -85,B 0,C 180,E1 29379.328,E2 29379.328} C_VEL
LIN {X 0,Y 630.466,Z 352.894,A -85,B 0,C 180,E1 29377.949,E2 29377.949} C_VEL
LIN {X 0,Y 626.956,Z 347.78,A -85,B 0,C 180,E1 29377.419,E2 29377.419} C_VEL
LIN {X 0,Y 621.158,Z 336.089,A -85,B 0,C 180,E1 29375.622,E2 29375.622} C_VEL
LIN {X 0,Y 619.355,Z 332.287,A -85,B 0,C 180,E1 29375.024,E2 29375.024} C_VEL
LIN {X 0,Y 617.337,Z 328.827,A -85,B 0,C 180,E1 29374.421,E2 29374.421} C_VEL
LIN {X 0,Y 617.009,Z 327.341,A -85,B 0,C 180,E1 29374.217,E2 29374.217} C_VEL
LIN {X 0,Y 616.975,Z 327.365,A -85,B 0,C 180,E1 29371.13,E2 29371.13} C_VEL
LIN {X 0,Y 617.016,Z 327.366,A -85,B 0,C 180,E1 29368.031,E2 29368.031} C_VEL
LIN {X 0,Y 616.967,Z 327.344,A -85,B 0,C 180,E1 29364.921,E2 29364.921} C_VEL
LIN {X 0,Y 617.016,Z 327.362,A -85,B 0,C 180,E1 29361.884,E2 29361.884} C_VEL
LIN {X 0,Y 616.965,Z 327.363,A -85,B 0,C 180,E1 29358.815,E2 29358.815} C_VEL
LIN {X 0,Y 617.014,Z 327.343,A -85,B 0,C 180,E1 29355.728,E2 29355.728} C_VEL
LIN {X 0,Y 616.96,Z 327.377,A -85,B 0,C 180,E1 29352.638,E2 29352.638} C_VEL
LIN {X 0,Y 617.012,Z 327.337,A -85,B 0,C 180,E1 29349.609,E2 29349.609} C_VEL
LIN {X 0,Y 616.956,Z 327.378,A -85,B 0,C 180,E1 29346.514,E2 29346.514} C_VEL
LIN {X 0,Y 617.011,Z 327.335,A -85,B 0,C 180,E1 29343.422,E2 29343.422} C_VEL
LIN {X 0,Y 616.949,Z 327.379,A -85,B 0,C 180,E1 29340.371,E2 29340.371} C_VEL
LIN {X 0,Y 617.004,Z 327.336,A -85,B 0,C 180,E1 29337.399,E2 29337.399} C_VEL
LIN {X 0,Y 616.945,Z 327.38,A -85,B 0,C 180,E1 29334.315,E2 29334.315} C_VEL
LIN {X 0,Y 616.971,Z 327.343,A -85,B 0,C 180,E1 29331.519,E2 29331.519} C_VEL
LIN {X 0,Y 616.944,Z 327.381,A -85,B 0,C 180,E1 29328.312,E2 29328.312} C_VEL
LIN {X 0,Y 616.95,Z 327.345,A -85,B 0,C 180,E1 29325.547,E2 29325.547} C_VEL
LIN {X 0,Y 616.945,Z 327.381,A -85,B 0,C 180,E1 29322.26,E2 29322.26} C_VEL
LIN {X 0,Y 616.934,Z 327.343,A -85,B 0,C 180,E1 29319.508,E2 29319.508} C_VEL
LIN {X 0,Y 616.953,Z 327.375,A -85,B 0,C 180,E1 29316.299,E2 29316.299} C_VEL
LIN {X 0,Y 616.927,Z 327.357,A -85,B 0,C 180,E1 29313.461,E2 29313.461} C_VEL
LIN {X 0,Y 616.971,Z 327.348,A -85,B 0,C 180,E1 29310.376,E2 29310.376} C_VEL
LIN {X 0,Y 616.916,Z 327.386,A -85,B 0,C 180,E1 29307.555,E2 29307.555} C_VEL
LIN {X 0,Y 616.988,Z 327.349,A -85,B 0,C 180,E1 29304.537,E2 29304.537} C_VEL
LIN {X 0,Y 616.941,Z 327.574,A -85,B 0,C 180,E1 29303.658,E2 29303.658} C_VEL
LIN {X 0,Y 618.1,Z 330.692,A -85,B 0,C 180,E1 29303.451,E2 29303.451} C_VEL
LIN {X 0,Y 620.746,Z 333.25,A -85,B 0,C 180,E1 29303.071,E2 29303.071} C_VEL
LIN {X 0,Y 621.615,Z 334.298,A -85,B 0,C 180,E1 29302.944,E2 29302.944} C_VEL
LIN {X 0,Y 624.325,Z 338.127,A -85,B 0,C 180,E1 29302.541,E2 29302.541} C_VEL
LIN {X 0,Y 625.964,Z 339.97,A -85,B 0,C 180,E1 29302.31,E2 29302.31} C_VEL
LIN {X 0,Y 629.219,Z 344.209,A -85,B 0,C 180,E1 29301.847,E2 29301.847} C_VEL
LIN {X 0,Y 635.275,Z 352.15,A -85,B 0,C 180,E1 29301.01,E2 29301.01} C_VEL
LIN {X 0,Y 645.89,Z 366.136,A -85,B 0,C 180,E1 29299.613,E2 29299.613} C_VEL
LIN {X 0,Y 655.156,Z 379.241,A -85,B 0,C 180,E1 29298.446,E2 29298.446} C_VEL
LIN {X 0,Y 656.048,Z 380.85,A -85,B 0,C 180,E1 29298.332,E2 29298.332} C_VEL
LIN {X 0,Y 654.312,Z 458.951,A -85,B 0,C 180,E1 29297.246,E2 29297.246} C_VEL
LIN {X 0,Y 653.478,Z 466.655,A -85,B 0,C 180,E1 29297.203,E2 29297.203} C_VEL
LIN {X 0,Y 648.749,Z 487.329,A -85,B 0,C 180,E1 29297.327,E2 29297.327} C_VEL
LIN {X 0,Y 648.081,Z 493.94,A -85,B 0,C 180,E1 29297.285,E2 29297.285} C_VEL
LIN {X 0,Y 643.293,Z 710.545,A -85,B 0,C 180,E1 29294.325,E2 29294.325} C_VEL
LIN {X 0,Y 641.272,Z 798.391,A -85,B 0,C 180,E1 29293.129,E2 29293.129} C_VEL
LIN {X 0,Y 639.997,Z 825.882,A -85,B 0,C 180,E1 29292.62,E2 29292.62} C_VEL
LIN {X 0,Y 638.311,Z 851.585,A -85,B 0,C 180,E1 29291.967,E2 29291.967} C_VEL
LIN {X 0,Y 636.68,Z 873.014,A -85,B 0,C 180,E1 29291.298,E2 29291.298} C_VEL
LIN {X 0,Y 634.97,Z 892.901,A -85,B 0,C 180,E1 29290.566,E2 29290.566} C_VEL
LIN {X 0,Y 632.853,Z 915.388,A -85,B 0,C 180,E1 29289.605,E2 29289.605} C_VEL
LIN {X 0,Y 630.159,Z 941.546,A -85,B 0,C 180,E1 29288.287,E2 29288.287} C_VEL
LIN {X 0,Y 627.817,Z 962.397,A -85,B 0,C 180,E1 29287.068,E2 29287.068} C_VEL
LIN {X 0,Y 625.666,Z 980.865,A -85,B 0,C 180,E1 29285.857,E2 29285.857} C_VEL
LIN {X 0,Y 623.421,Z 999.81,A -85,B 0,C 180,E1 29284.473,E2 29284.473} C_VEL
LIN {X 0,Y 620.78,Z 1021.939,A -85,B 0,C 180,E1 29282.654,E2 29282.654} C_VEL
LIN {X 0,Y 618.413,Z 1041.363,A -85,B 0,C 180,E1 29280.832,E2 29280.832} C_VEL
LIN {X 0,Y 616.552,Z 1057.379,A -85,B 0,C 180,E1 29279.164,E2 29279.164} C_VEL
LIN {X 0,Y 614.613,Z 1075.24,A -85,B 0,C 180,E1 29277.097,E2 29277.097} C_VEL
LIN {X 0,Y 612.779,Z 1092.683,A -85,B 0,C 180,E1 29274.793,E2 29274.793} C_VEL
LIN {X 0,Y 611.507,Z 1106.097,A -85,B 0,C 180,E1 29272.8,E2 29272.8} C_VEL
LIN {X 0,Y 610.328,Z 1120.339,A -85,B 0,C 180,E1 29270.423,E2 29270.423} C_VEL
LIN {X 0,Y 609.403,Z 1132.944,A -85,B 0,C 180,E1 29267.966,E2 29267.966} C_VEL
LIN {X 0,Y 608.859,Z 1142.121,A -85,B 0,C 180,E1 29265.917,E2 29265.917} C_VEL
LIN {X 0,Y 608.471,Z 1150.056,A -85,B 0,C 180,E1 29263.881,E2 29263.881} C_VEL
LIN {X 0,Y 608.195,Z 1157.753,A -85,B 0,C 180,E1 29261.57,E2 29261.57} C_VEL
LIN {X 0,Y 608.015,Z 1164.592,A -85,B 0,C 180,E1 29258.988,E2 29258.988} C_VEL
LIN {X 0,Y 607.942,Z 1169.367,A -85,B 0,C 180,E1 29256.581,E2 29256.581} C_VEL
LIN {X 0,Y 607.918,Z 1172.634,A -85,B 0,C 180,E1 29254.244,E2 29254.244} C_VEL
LIN {X 0,Y 607.907,Z 1174.59,A -85,B 0,C 180,E1 29251.697,E2 29251.697} C_VEL
LIN {X 0,Y 607.895,Z 1174.86,A -85,B 0,C 180,E1 29249.34,E2 29249.34} C_VEL
LIN {X 0,Y 607.911,Z 1173.963,A -85,B 0,C 180,E1 29247.172,E2 29247.172} C_VEL
LIN {X 0,Y 607.922,Z 1171.72,A -85,B 0,C 180,E1 29244.905,E2 29244.905} C_VEL
LIN {X 0,Y 607.963,Z 1167.635,A -85,B 0,C 180,E1 29242.345,E2 29242.345} C_VEL
LIN {X 0,Y 608.076,Z 1161.986,A -85,B 0,C 180,E1 29239.867,E2 29239.867} C_VEL
LIN {X 0,Y 608.268,Z 1155.244,A -85,B 0,C 180,E1 29237.538,E2 29237.538} C_VEL
LIN {X 0,Y 608.665,Z 1146.287,A -85,B 0,C 180,E1 29235.005,E2 29235.005} C_VEL
LIN {X 0,Y 609.26,Z 1135.375,A -85,B 0,C 180,E1 29232.462,E2 29232.462} C_VEL
LIN {X 0,Y 609.973,Z 1124.992,A -85,B 0,C 180,E1 29230.365,E2 29230.365} C_VEL
LIN {X 0,Y 610.926,Z 1112.795,A -85,B 0,C 180,E1 29228.191,E2 29228.191} C_VEL
LIN {X 0,Y 612.374,Z 1096.799,A -85,B 0,C 180,E1 29225.704,E2 29225.704} C_VEL
LIN {X 0,Y 613.835,Z 1082.184,A -85,B 0,C 180,E1 29223.701,E2 29223.701} C_VEL
LIN {X 0,Y 615.508,Z 1066.659,A -85,B 0,C 180,E1 29221.79,E2 29221.79} C_VEL
LIN {X 0,Y 617.898,Z 1045.992,A -85,B 0,C 180,E1 29219.541,E2 29219.541} C_VEL
LIN {X 0,Y 619.936,Z 1028.597,A -85,B 0,C 180,E1 29217.862,E2 29217.862} C_VEL
LIN {X 0,Y 622.051,Z 1010.9,A -85,B 0,C 180,E1 29216.321,E2 29216.321} C_VEL
LIN {X 0,Y 624.78,Z 988.7,A -85,B 0,C 180,E1 29214.597,E2 29214.597} C_VEL
LIN {X 0,Y 627.4,Z 966.083,A -85,B 0,C 180,E1 29213.072,E2 29213.072} C_VEL
LIN {X 0,Y 629.504,Z 947.446,A -85,B 0,C 180,E1 29211.956,E2 29211.956} C_VEL
LIN {X 0,Y 631.538,Z 928.466,A -85,B 0,C 180,E1 29210.941,E2 29210.941} C_VEL
LIN {X 0,Y 633.584,Z 908.068,A -85,B 0,C 180,E1 29209.979,E2 29209.979} C_VEL
LIN {X 0,Y 635.939,Z 882.61,A -85,B 0,C 180,E1 29208.943,E2 29208.943} C_VEL
LIN {X 0,Y 637.968,Z 856.338,A -85,B 0,C 180,E1 29208.08,E2 29208.08} C_VEL
LIN {X 0,Y 639.432,Z 834.476,A -85,B 0,C 180,E1 29207.494,E2 29207.494} C_VEL
LIN {X 0,Y 640.647,Z 812.416,A -85,B 0,C 180,E1 29207.022,E2 29207.022} C_VEL
LIN {X 0,Y 641.75,Z 784.837,A -85,B 0,C 180,E1 29206.581,E2 29206.581} C_VEL
LIN {X 0,Y 646.583,Z 560.106,A -85,B 0,C 180,E1 29203.539,E2 29203.539} C_VEL
LIN {X 0,Y 650.59,Z 384.361,A -85,B 0,C 180,E1 29201.088,E2 29201.088} C_VEL
LIN {X 0,Y 637.854,Z 366.542,A -85,B 0,C 180,E1 29199.44,E2 29199.44} C_VEL
LIN {X 0,Y 625.845,Z 350.856,A -85,B 0,C 180,E1 29197.786,E2 29197.786} C_VEL
LIN {X 0,Y 621.131,Z 344.899,A -85,B 0,C 180,E1 29197.105,E2 29197.105} C_VEL
LIN {X 0,Y 617.43,Z 340.07,A -85,B 0,C 180,E1 29196.552,E2 29196.552} C_VEL
LIN {X 0,Y 614.443,Z 336.735,A -85,B 0,C 180,E1 29196.107,E2 29196.107} C_VEL
LIN {X 0,Y 613.14,Z 334.405,A -85,B 0,C 180,E1 29195.892,E2 29195.892} C_VEL
LIN {X 0,Y 610.477,Z 332.003,A -85,B 0,C 180,E1 29195.495,E2 29195.495} C_VEL
LIN {X 0,Y 609.119,Z 328.913,A -85,B 0,C 180,E1 29195.252,E2 29195.252} C_VEL
LIN {X 0,Y 609.022,Z 328.336,A -85,B 0,C 180,E1 29195.224,E2 29195.224} C_VEL
LIN {X 0,Y 608.973,Z 328.376,A -85,B 0,C 180,E1 29192.251,E2 29192.251} C_VEL
LIN {X 0,Y 609.038,Z 328.342,A -85,B 0,C 180,E1 29189.146,E2 29189.146} C_VEL
LIN {X 0,Y 608.975,Z 328.342,A -85,B 0,C 180,E1 29186.211,E2 29186.211} C_VEL
LIN {X 0,Y 609.06,Z 328.367,A -85,B 0,C 180,E1 29183.102,E2 29183.102} C_VEL
LIN {X 0,Y 608.98,Z 328.331,A -85,B 0,C 180,E1 29180.17,E2 29180.17} C_VEL
LIN {X 0,Y 609.061,Z 328.363,A -85,B 0,C 180,E1 29177.17,E2 29177.17} C_VEL
LIN {X 0,Y 608.99,Z 328.335,A -85,B 0,C 180,E1 29174.161,E2 29174.161} C_VEL
LIN {X 0,Y 609.035,Z 328.366,A -85,B 0,C 180,E1 29171.266,E2 29171.266} C_VEL
LIN {X 0,Y 609,Z 328.335,A -85,B 0,C 180,E1 29168.108,E2 29168.108} C_VEL
LIN {X 0,Y 609.017,Z 328.37,A -85,B 0,C 180,E1 29165.37,E2 29165.37} C_VEL
LIN {X 0,Y 609.011,Z 328.332,A -85,B 0,C 180,E1 29162.07,E2 29162.07} C_VEL
LIN {X 0,Y 609.024,Z 328.369,A -85,B 0,C 180,E1 29159.247,E2 29159.247} C_VEL
LIN {X 0,Y 609.02,Z 328.331,A -85,B 0,C 180,E1 29155.952,E2 29155.952} C_VEL
LIN {X 0,Y 609.035,Z 328.363,A -85,B 0,C 180,E1 29153.022,E2 29153.022} C_VEL
LIN {X 0,Y 609.024,Z 328.337,A -85,B 0,C 180,E1 29149.787,E2 29149.787} C_VEL
LIN {X 0,Y 609.048,Z 328.351,A -85,B 0,C 180,E1 29146.809,E2 29146.809} C_VEL
LIN {X 0,Y 609.031,Z 328.351,A -85,B 0,C 180,E1 29143.597,E2 29143.597} C_VEL
LIN {X 0,Y 609.064,Z 328.33,A -85,B 0,C 180,E1 29140.533,E2 29140.533} C_VEL
LIN {X 0,Y 609.031,Z 328.366,A -85,B 0,C 180,E1 29137.305,E2 29137.305} C_VEL
LIN {X 0,Y 609.073,Z 328.328,A -85,B 0,C 180,E1 29134.212,E2 29134.212} C_VEL
LIN {X 0,Y 609.032,Z 328.341,A -85,B 0,C 180,E1 29131.139,E2 29131.139} C_VEL
LIN {X 0,Y 609.076,Z 328.364,A -85,B 0,C 180,E1 29128.071,E2 29128.071} C_VEL
LIN {X 0,Y 609.064,Z 328.524,A -85,B 0,C 180,E1 29126.719,E2 29126.719} C_VEL
LIN {X 0,Y 610.507,Z 332.002,A -85,B 0,C 180,E1 29126.161,E2 29126.161} C_VEL
LIN {X 0,Y 611.678,Z 333.968,A -85,B 0,C 180,E1 29125.803,E2 29125.803} C_VEL
LIN {X 0,Y 614.285,Z 339.279,A -85,B 0,C 180,E1 29124.929,E2 29124.929} C_VEL
LIN {X 0,Y 618.666,Z 347.822,A -85,B 0,C 180,E1 29123.562,E2 29123.562} C_VEL
LIN {X 0,Y 630.319,Z 364.077,A -85,B 0,C 180,E1 29121.868,E2 29121.868} C_VEL
LIN {X 0,Y 643.314,Z 382.84,A -85,B 0,C 180,E1 29120.108,E2 29120.108} C_VEL
LIN {X 0,Y 650.971,Z 394.486,A -85,B 0,C 180,E1 29119.123,E2 29119.123} C_VEL
LIN {X 0,Y 646.286,Z 600.291,A -85,B 0,C 180,E1 29116.272,E2 29116.272} C_VEL
LIN {X 0,Y 641.574,Z 820.021,A -85,B 0,C 180,E1 29113.298,E2 29113.298} C_VEL
LIN {X 0,Y 640.582,Z 843.71,A -85,B 0,C 180,E1 29112.908,E2 29112.908} C_VEL
LIN {X 0,Y 639.37,Z 865.449,A -85,B 0,C 180,E1 29112.437,E2 29112.437} C_VEL
LIN {X 0,Y 637.845,Z 888.081,A -85,B 0,C 180,E1 29111.824,E2 29111.824} C_VEL
LIN {X 0,Y 635.602,Z 916.168,A -85,B 0,C 180,E1 29110.874,E2 29110.874} C_VEL
LIN {X 0,Y 633.472,Z 939.121,A -85,B 0,C 180,E1 29109.93,E2 29109.93} C_VEL
LIN {X 0,Y 631.438,Z 959.397,A -85,B 0,C 180,E1 29108.967,E2 29108.967} C_VEL
LIN {X 0,Y 629.282,Z 979.446,A -85,B 0,C 180,E1 29107.887,E2 29107.887} C_VEL
LIN {X 0,Y 626.559,Z 1003.45,A -85,B 0,C 180,E1 29106.415,E2 29106.415} C_VEL
LIN {X 0,Y 623.934,Z 1025.29,A -85,B 0,C 180,E1 29104.864,E2 29104.864} C_VEL
LIN {X 0,Y 621.763,Z 1043.425,A -85,B 0,C 180,E1 29103.422,E2 29103.422} C_VEL
LIN {X 0,Y 619.645,Z 1061.276,A -85,B 0,C 180,E1 29101.846,E2 29101.846} C_VEL
LIN {X 0,Y 617.112,Z 1082.695,A -85,B 0,C 180,E1 29099.719,E2 29099.719} C_VEL
LIN {X 0,Y 615.205,Z 1099.307,A -85,B 0,C 180,E1 29097.851,E2 29097.851} C_VEL
LIN {X 0,Y 613.573,Z 1114.932,A -85,B 0,C 180,E1 29095.895,E2 29095.895} C_VEL
LIN {X 0,Y 611.896,Z 1131.901,A -85,B 0,C 180,E1 29093.497,E2 29093.497} C_VEL
LIN {X 0,Y 610.754,Z 1144.86,A -85,B 0,C 180,E1 29091.412,E2 29091.412} C_VEL
LIN {X 0,Y 609.862,Z 1156.304,A -85,B 0,C 180,E1 29089.34,E2 29089.34} C_VEL
LIN {X 0,Y 609.085,Z 1168.202,A -85,B 0,C 180,E1 29086.891,E2 29086.891} C_VEL
LIN {X 0,Y 608.568,Z 1178.091,A -85,B 0,C 180,E1 29084.462,E2 29084.462} C_VEL
LIN {X 0,Y 608.253,Z 1185.489,A -85,B 0,C 180,E1 29082.339,E2 29082.339} C_VEL
LIN {X 0,Y 608.07,Z 1192.121,A -85,B 0,C 180,E1 29080.038,E2 29080.038} C_VEL
LIN {X 0,Y 607.963,Z 1197.908,A -85,B 0,C 180,E1 29077.465,E2 29077.465} C_VEL
LIN {X 0,Y 607.924,Z 1201.78,A -85,B 0,C 180,E1 29075.001,E2 29075.001} C_VEL
LIN {X 0,Y 607.912,Z 1203.998,A -85,B 0,C 180,E1 29072.734,E2 29072.734} C_VEL
LIN {X 0,Y 607.893,Z 1204.894,A -85,B 0,C 180,E1 29070.471,E2 29070.471} C_VEL
LIN {X 0,Y 607.911,Z 1204.382,A -85,B 0,C 180,E1 29067.832,E2 29067.832} C_VEL
LIN {X 0,Y 607.914,Z 1202.234,A -85,B 0,C 180,E1 29065.377,E2 29065.377} C_VEL
LIN {X 0,Y 607.944,Z 1198.913,A -85,B 0,C 180,E1 29063.104,E2 29063.104} C_VEL
LIN {X 0,Y 608.042,Z 1193.595,A -85,B 0,C 180,E1 29060.535,E2 29060.535} C_VEL
LIN {X 0,Y 608.218,Z 1186.572,A -85,B 0,C 180,E1 29058.005,E2 29058.005} C_VEL
LIN {X 0,Y 608.513,Z 1179.16,A -85,B 0,C 180,E1 29055.829,E2 29055.829} C_VEL
LIN {X 0,Y 608.944,Z 1170.674,A -85,B 0,C 180,E1 29053.694,E2 29053.694} C_VEL
LIN {X 0,Y 609.729,Z 1158.367,A -85,B 0,C 180,E1 29051.053,E2 29051.053} C_VEL
LIN {X 0,Y 610.664,Z 1146.01,A -85,B 0,C 180,E1 29048.786,E2 29048.786} C_VEL
LIN {X 0,Y 611.78,Z 1133.191,A -85,B 0,C 180,E1 29046.702,E2 29046.702} C_VEL
LIN {X 0,Y 613.496,Z 1115.702,A -85,B 0,C 180,E1 29044.205,E2 29044.205} C_VEL
LIN {X 0,Y 615.166,Z 1099.687,A -85,B 0,C 180,E1 29042.194,E2 29042.194} C_VEL
LIN {X 0,Y 616.995,Z 1083.602,A -85,B 0,C 180,E1 29040.379,E2 29040.379} C_VEL
LIN {X 0,Y 619.561,Z 1062.029,A -85,B 0,C 180,E1 29038.223,E2 29038.223} C_VEL
LIN {X 0,Y 621.693,Z 1044.052,A -85,B 0,C 180,E1 29036.631,E2 29036.631} C_VEL
LIN {X 0,Y 623.822,Z 1026.229,A -85,B 0,C 180,E1 29035.208,E2 29035.208} C_VEL
LIN {X 0,Y 626.365,Z 1004.911,A -85,B 0,C 180,E1 29033.685,E2 29033.685} C_VEL
LIN {X 0,Y 629.183,Z 980.345,A -85,B 0,C 180,E1 29032.164,E2 29032.164} C_VEL
LIN {X 0,Y 631.406,Z 959.706,A -85,B 0,C 180,E1 29031.048,E2 29031.048} C_VEL
LIN {X 0,Y 633.39,Z 939.909,A -85,B 0,C 180,E1 29030.105,E2 29030.105} C_VEL
LIN {X 0,Y 635.448,Z 917.788,A -85,B 0,C 180,E1 29029.189,E2 29029.189} C_VEL
LIN {X 0,Y 637.733,Z 889.776,A -85,B 0,C 180,E1 29028.226,E2 29028.226} C_VEL
LIN {X 0,Y 639.334,Z 866.07,A -85,B 0,C 180,E1 29027.578,E2 29027.578} C_VEL
LIN {X 0,Y 640.554,Z 844.303,A -85,B 0,C 180,E1 29027.103,E2 29027.103} C_VEL
LIN {X 0,Y 641.526,Z 821.332,A -85,B 0,C 180,E1 29026.721,E2 29026.721} C_VEL
LIN {X 0,Y 646.235,Z 602.686,A -85,B 0,C 180,E1 29023.761,E2 29023.761} C_VEL
LIN {X 0,Y 650.93,Z 396.261,A -85,B 0,C 180,E1 29020.902,E2 29020.902} C_VEL
LIN {X 0,Y 650.812,Z 393.99,A -85,B 0,C 180,E1 29020.853,E2 29020.853} C_VEL
LIN {X 0,Y 634.447,Z 369.819,A -85,B 0,C 180,E1 29018.703,E2 29018.703} C_VEL
LIN {X 0,Y 621.432,Z 351.589,A -85,B 0,C 180,E1 29016.853,E2 29016.853} C_VEL
LIN {X 0,Y 618.436,Z 347.33,A -85,B 0,C 180,E1 29016.376,E2 29016.376} C_VEL
LIN {X 0,Y 614.846,Z 340.448,A -85,B 0,C 180,E1 29015.262,E2 29015.262} C_VEL
LIN {X 0,Y 613.121,Z 336.94,A -85,B 0,C 180,E1 29014.692,E2 29014.692} C_VEL
LIN {X 0,Y 611.194,Z 332.833,A -85,B 0,C 180,E1 29014.021,E2 29014.021} C_VEL
LIN {X 0,Y 609.365,Z 329.775,A -85,B 0,C 180,E1 29013.459,E2 29013.459} C_VEL
LIN {X 0,Y 609.038,Z 328.335,A -85,B 0,C 180,E1 29013.254,E2 29013.254} C_VEL
LIN {X 0,Y 609.074,Z 328.327,A -85,B 0,C 180,E1 29010.156,E2 29010.156} C_VEL
LIN {X 0,Y 609.035,Z 328.362,A -85,B 0,C 180,E1 29007.05,E2 29007.05} C_VEL
LIN {X 0,Y 609.075,Z 328.344,A -85,B 0,C 180,E1 29003.884,E2 29003.884} C_VEL
LIN {X 0,Y 609.026,Z 328.332,A -85,B 0,C 180,E1 29000.871,E2 29000.871} C_VEL
LIN {X 0,Y 609.078,Z 328.36,A -85,B 0,C 180,E1 28997.779,E2 28997.779} C_VEL
LIN {X 0,Y 609.017,Z 328.328,A -85,B 0,C 180,E1 28994.646,E2 28994.646} C_VEL
LIN {X 0,Y 609.079,Z 328.362,A -85,B 0,C 180,E1 28991.553,E2 28991.553} C_VEL
LIN {X 0,Y 609.014,Z 328.332,A -85,B 0,C 180,E1 28988.497,E2 28988.497} C_VEL
LIN {X 0,Y 609.079,Z 328.359,A -85,B 0,C 180,E1 28985.464,E2 28985.464} C_VEL
LIN {X 0,Y 609.009,Z 328.334,A -85,B 0,C 180,E1 28982.352,E2 28982.352} C_VEL
LIN {X 0,Y 609.079,Z 328.355,A -85,B 0,C 180,E1 28979.248,E2 28979.248} C_VEL
LIN {X 0,Y 609.003,Z 328.337,A -85,B 0,C 180,E1 28976.14,E2 28976.14} C_VEL
LIN {X 0,Y 609.073,Z 328.352,A -85,B 0,C 180,E1 28973.022,E2 28973.022} C_VEL
LIN {X 0,Y 608.998,Z 328.34,A -85,B 0,C 180,E1 28969.977,E2 28969.977} C_VEL
LIN {X 0,Y 609.07,Z 328.349,A -85,B 0,C 180,E1 28966.906,E2 28966.906} C_VEL
LIN {X 0,Y 608.992,Z 328.345,A -85,B 0,C 180,E1 28963.988,E2 28963.988} C_VEL
LIN {X 0,Y 609.059,Z 328.345,A -85,B 0,C 180,E1 28961.012,E2 28961.012} C_VEL
